KUKA KRL program: ps_r5_l_resp1_c1_mod.src, ps_r5_l_resp1_c1_mod.dat

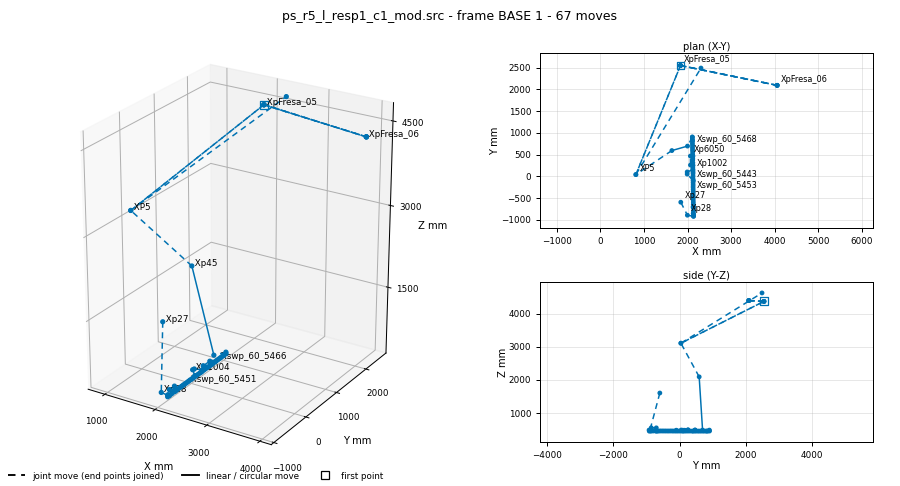
[picture p0: tool path of ps_r5_l_resp1_c1_mod.src in frame BASE 1, 67 of 69 moves have a stored position in this frame; points joined in program order, loops and branches not executed]
--- ps_r5_l_resp1_c1_mod.src ---
&ACCESS RVO1
&REL 40
&COMMENT C1 Respot LTA/LTB/MGS/MGSB
&PARAM DISKPATH = KRC:\R1\Program\SOLDA LTC
DEF ps_r5_l_resp1_c1_mod( )
;FOLD INI
  ;FOLD BASISTECH INI
    GLOBAL INTERRUPT DECL 3 WHEN $STOPMESS==TRUE DO IR_STOPM ( )
    INTERRUPT ON 3
    BAS (#INITMOV,0 )
  ;ENDFOLD (BASISTECH INI)
;FOLD SPOTTECH INI
USERSPOT(#INIT)
;ENDFOLD (SPOTTECH INI)
;FOLD GRIPPERTECH INI

;ENDFOLD (GRIPPERTECH INI)
  ;FOLD USER INI
    ;Make your modifications here

     ;FOLD COLLISION_V_3.01 INI ;%{E}
        IF (COLLISION_DATA[1].I_NR>0) THEN
          GLOBAL INTERRUPT DECL 21 WHEN $IN[COLLISION_DATA[1].I_NR]==FALSE DO COLLSTOP (1,0 )
        ENDIF
        IF (COLLISION_DATA[2].I_NR>0) THEN
          GLOBAL INTERRUPT DECL 22 WHEN $IN[COLLISION_DATA[2].I_NR]==FALSE DO COLLSTOP (2,0 )
        ENDIF
        IF (COLLISION_DATA[3].I_NR>0) THEN
          GLOBAL INTERRUPT DECL 23 WHEN $IN[COLLISION_DATA[3].I_NR]==FALSE DO COLLSTOP (3,0 )
        ENDIF
        IF (COLLISION_DATA[4].I_NR>0) THEN
          GLOBAL INTERRUPT DECL 24 WHEN $IN[COLLISION_DATA[4].I_NR]==FALSE DO COLLSTOP (4,0 )
        ENDIF
     ;ENDFOLD (Collision)

  ;ENDFOLD (USER INI)
;ENDFOLD (INI)

; Caracterização dos meios de produção: P13.060-R5
; Versão atual: 17/07/2013 Nome: Solda Respot C1
; Change: LTA/LTB/MGS/MGSB

chk_w2_wechs_ok ( )           ; VERIFICAÇÃO DE FERRAMENA: C1

;FOLD PTP HOME2 Vel=100 % DEFAULT;%{PE}%R 8.2.20,%MKUKATPBASIS,%CMOVE,%VPTP,%P 1:PTP, 2:HOME2, 3:, 5:100, 7:DEFAULT
$BWDSTART=FALSE
PDAT_ACT=PDEFAULT
FDAT_ACT=FHOME2
BAS(#PTP_PARAMS,100)
PTP XHOME2
;ENDFOLD

IF(NOT(GHOST())) THEN
IF MaxStandMenge (1) THEN
 MaxStandmengeErreicht (1)
ENDIF

IF Elektrodenwechsel (1) THEN
;FOLD PTP pFresa_05 CONT Vel=100 % PDAT40 Tool[2]:Gun C1 Base[1]:Actros;%{PE}%R 8.2.20,%MKUKATPBASIS,%CMOVE,%VPTP,%P 1:PTP, 2:pFresa_05, 3:C_DIS, 5:100, 7:PDAT40
$BWDSTART=FALSE
PDAT_ACT=PPDAT40
FDAT_ACT=FpFresa_05
BAS(#PTP_PARAMS,100)
PTP XpFresa_05 C_DIS
;ENDFOLD
;FOLD PULSE 168 'DOCK 1 Fechar Proteção' State=TRUE Time=1 sec;%{PE}%R 8.2.20,%MKUKATPBASIS,%COUT,%VPULSE,%P 2:168, 3:DOCK 1 Fechar Proteção, 5:TRUE, 6:, 8:1
PULSE($OUT[168], TRUE,1)
;ENDFOLD
;FOLD WAIT FOR ( IN 166 'DOCK 1 Proteção Fechada' );%{PE}%R 8.2.20,%MKUKATPBASIS,%CEXT_WAIT_FOR,%VEXT_WAIT_FOR,%P 2:, 4:, 5:$IN, 6:166, 7:DOCK 1 Proteção Fechada, 9:
WAIT FOR  ( $IN[166] )
;ENDFOLD
;FOLD PTP pFresa_06 CONT Vel=100 % PDAT41 Tool[2]:Gun C1 Base[1]:Actros;%{PE}%R 8.2.20,%MKUKATPBASIS,%CMOVE,%VPTP,%P 1:PTP, 2:pFresa_06, 3:C_DIS, 5:100, 7:PDAT41
$BWDSTART=FALSE
PDAT_ACT=PPDAT41
FDAT_ACT=FpFresa_06
BAS(#PTP_PARAMS,100)
PTP XpFresa_06 C_DIS
;ENDFOLD
 e_Fraes_2 ()
;FOLD PTP pFresa_07 CONT Vel=100 % PDAT42 Tool[2]:Gun C1 Base[1]:Actros;%{PE}%R 8.2.20,%MKUKATPBASIS,%CMOVE,%VPTP,%P 1:PTP, 2:pFresa_07, 3:C_DIS, 5:100, 7:PDAT42
$BWDSTART=FALSE
PDAT_ACT=PPDAT42
FDAT_ACT=FpFresa_07
BAS(#PTP_PARAMS,100)
PTP XpFresa_07 C_DIS
;ENDFOLD
;FOLD PTP pFresa_08 CONT Vel=100 % PDAT43 Tool[2]:Gun C1 Base[1]:Actros;%{PE}%R 8.2.20,%MKUKATPBASIS,%CMOVE,%VPTP,%P 1:PTP, 2:pFresa_08, 3:C_DIS, 5:100, 7:PDAT43
$BWDSTART=FALSE
PDAT_ACT=PPDAT43
FDAT_ACT=FpFresa_08
BAS(#PTP_PARAMS,100)
PTP XpFresa_08 C_DIS
;ENDFOLD
ENDIF
ENDIF
;FOLD PTP HOME2 Vel=100 % DEFAULT;%{PE}%R 8.2.20,%MKUKATPBASIS,%CMOVE,%VPTP,%P 1:PTP, 2:HOME2, 3:, 5:100, 7:DEFAULT
$BWDSTART=FALSE
PDAT_ACT=PDEFAULT
FDAT_ACT=FHOME2
BAS(#PTP_PARAMS,100)
PTP XHOME2
;ENDFOLD

;FOLD OUT 3339 'R5 SOLDANDO' State=TRUE ;%{PE}%R 8.2.20,%MKUKATPBASIS,%COUT,%VOUTX,%P 2:3339, 3:R5 SOLDANDO, 5:TRUE, 6:
$OUT[3339]=TRUE
;ENDFOLD
;FOLD OUT 3340 'locking-signal PLC' State=FALSE ;%{PE}%R 8.2.20,%MKUKATPBASIS,%COUT,%VOUTX,%P 2:3340, 3:locking-signal PLC, 5:FALSE, 6:
$OUT[3340]=FALSE
;ENDFOLD

;FOLD PTP p27 CONT Vel=100 % P_OLP2 Tool[2]:Gun C1 Base[1]:Actros;%{PE}%R 8.2.20,%MKUKATPBASIS,%CMOVE,%VPTP,%P 1:PTP, 2:p27, 3:C_DIS, 5:100, 7:P_OLP2
$BWDSTART=FALSE
PDAT_ACT=PP_OLP2
FDAT_ACT=Fp27
BAS(#PTP_PARAMS,100)
PTP Xp27 C_DIS
;ENDFOLD
;FOLD PTP p28 CONT Vel=100 % P_OLP3 Tool[2]:Gun C1 Base[1]:Actros;%{PE}%R 8.2.20,%MKUKATPBASIS,%CMOVE,%VPTP,%P 1:PTP, 2:p28, 3:C_DIS, 5:100, 7:P_OLP3
$BWDSTART=FALSE
PDAT_ACT=PP_OLP3
FDAT_ACT=Fp28
BAS(#PTP_PARAMS,100)
PTP Xp28 C_DIS
;ENDFOLD
;FOLD PTP p29 CONT Vel=100 % P_OLP4 Tool[2]:Gun C1 Base[1]:Actros;%{PE}%R8.2,%MKUKATPBASIS,%CMOVE,%VPTP,%P 1:PTP, 2:p29, 3:C_DIS, 5:100, 7:P_OLP4
$BWDSTART = FALSE
PDAT_ACT= PP_OLP4
FDAT_ACT= Fp29
BAS(#PTP_PARAMS,100)
PTP Xp29 C_DIS
;ENDFOLD

;FOLD ; SWP_60_5475;%{PE}%R 8.2.20,%MKUKATPBASIS,%CCOMMENT,%VNORMAL,%P 2:SWP_60_5475
;ENDFOLD
;FOLD PTP swp_60_5475 PDAT1 SPOT Gun=1 RETR OPN PgNo1=20 ACTIVE=1 Tool[2]:Gun C1 Base[1]:Actros;%{PE}%R 8.2.2,%MKUKATPSPOT,%CSPOT,%VPTP,%P 1:PTP, 2:swp_60_5475, 3:, 5:100, 7:PDAT1, 10:1, 12:#FIRST, 14:#OPN, 16:20, 18:1, 20:0, 22:0, 24:1, 25:NORMAL
$BWDSTART=FALSE
PDAT_ACT=PPDAT1
FDAT_ACT=Fswp_60_5475
BAS(#PTP_PARAMS,PPDAT1.VEL)
S_ACT.GUN=1
S_ACT.PAIR=SDEFAULT.PAIR
S_ACT.RETR=#OPN
S_ACT.CLO_TM=1
S_ACT.PGNO1=20
S_ACT.PGNO2=SDEFAULT.PGNO2
S_ACT.PRESS1=SDEFAULT.PRESS1
S_ACT.PRESS2=SDEFAULT.PRESS2
S_READY=FALSE
PTP Xswp_60_5475
USERSPOT(#SPOT, S_ACT)
WAIT FOR S_READY
;ENDFOLD
;FOLD PTP p6045 Vel=100 % PDAT48 Tool[2]:Gun C1 Base[1]:Actros;%{PE}%R 8.2.20,%MKUKATPBASIS,%CMOVE,%VPTP,%P 1:PTP, 2:p6045, 3:, 5:100, 7:PDAT48
$BWDSTART=FALSE
PDAT_ACT=PPDAT48
FDAT_ACT=Fp6045
BAS(#PTP_PARAMS,100)
PTP Xp6045
;ENDFOLD

;FOLD ; SWP_60_5473;%{PE}%R 8.2.20,%MKUKATPBASIS,%CCOMMENT,%VNORMAL,%P 2:SWP_60_5473
;ENDFOLD
;FOLD PTP swp_60_5473 PDAT2 SPOT Gun=1 RETR OPN PgNo1=21 ACTIVE=1 Tool[2]:Gun C1 Base[1]:Actros;%{PE}%R 8.2.2,%MKUKATPSPOT,%CSPOT,%VPTP,%P 1:PTP, 2:swp_60_5473, 3:, 5:100, 7:PDAT2, 10:1, 12:#FIRST, 14:#OPN, 16:21, 18:1, 20:0, 22:0, 24:1, 25:NORMAL
$BWDSTART=FALSE
PDAT_ACT=PPDAT2
FDAT_ACT=Fswp_60_5473
BAS(#PTP_PARAMS,PPDAT2.VEL)
S_ACT.GUN=1
S_ACT.PAIR=SDEFAULT.PAIR
S_ACT.RETR=#OPN
S_ACT.CLO_TM=1
S_ACT.PGNO1=21
S_ACT.PGNO2=SDEFAULT.PGNO2
S_ACT.PRESS1=SDEFAULT.PRESS1
S_ACT.PRESS2=SDEFAULT.PRESS2
S_READY=FALSE
PTP Xswp_60_5473
USERSPOT(#SPOT, S_ACT)
WAIT FOR S_READY
;ENDFOLD

; INSERCAO DO PONTO 60_5471 (ACTROS RETO_SEM BOLHA)
IF ($IN[3341]==TRUE) THEN

Wait for false
;FOLD ; Favor chamar a manutencao;%{PE}%R 8.2.20,%MKUKATPBASIS,%CCOMMENT,%VNORMAL,%P 2:Favor  chamar  a  manutencao
;ENDFOLD

;FOLD ; SWP_60_5471;%{PE}%R 8.2.20,%MKUKATPBASIS,%CCOMMENT,%VNORMAL,%P 2: SWP_60_5471
;ENDFOLD
;FOLD PTP swp_60_5477 P_OLP55 SPOT Gun=1 RETR OPN PgNo1=55 ACTIVE=1 Tool[2]:Gun C1 Base[1]:Actros;%{PE}%R 8.2.2,%MKUKATPSPOT,%CSPOT,%VPTP,%P 1:PTP, 2:swp_60_5477, 3:, 5:100, 7:P_OLP55, 10:1, 12:#FIRST, 14:#OPN, 16:55, 18:1, 20:1, 22:0, 24:1, 25:S_OLP1
$BWDSTART=FALSE
PDAT_ACT=PP_OLP55
FDAT_ACT=Fswp_60_5477
BAS(#PTP_PARAMS,PP_OLP55.VEL)
S_ACT.GUN=1
S_ACT.PAIR=SDEFAULT.PAIR
S_ACT.RETR=#OPN
S_ACT.CLO_TM=1
S_ACT.PGNO1=55
S_ACT.PGNO2=SDEFAULT.PGNO2
S_ACT.PRESS1=SDEFAULT.PRESS1
S_ACT.PRESS2=SDEFAULT.PRESS2
S_READY=FALSE
PTP Xswp_60_5477
USERSPOT(#SPOT, S_ACT)
WAIT FOR S_READY

;ENDFOLD
ENDIF

IF ($IN[3341]==FALSE) THEN
;FOLD PTP p30 CONT Vel=100 % P_OLP6 Tool[2]:Gun C1 Base[1]:Actros;%{PE}%R8.2,%MKUKATPBASIS,%CMOVE,%VPTP,%P 1:PTP, 2:p30, 3:C_DIS, 5:100, 7:P_OLP6
$BWDSTART = FALSE
PDAT_ACT= PP_OLP6
FDAT_ACT= Fp30
BAS(#PTP_PARAMS,100)
PTP Xp30 C_DIS
;ENDFOLD
;FOLD PTP p1005 CONT Vel=100 % DEFAULT Tool[2]:Gun C1 Base[1]:Actros;%{PE}%R 8.2.20,%MKUKATPBASIS,%CMOVE,%VPTP,%P 1:PTP, 2:p1005, 3:C_DIS, 5:100, 7:DEFAULT
$BWDSTART=FALSE
PDAT_ACT=PDEFAULT
FDAT_ACT=Fp1005
BAS(#PTP_PARAMS,100)
PTP Xp1005 C_DIS
;ENDFOLD
;FOLD PTP p31 CONT Vel=100 % P_OLP7 Tool[2]:Gun C1 Base[1]:Actros;%{PE}%R8.2,%MKUKATPBASIS,%CMOVE,%VPTP,%P 1:PTP, 2:p31, 3:C_DIS, 5:100, 7:P_OLP7
$BWDSTART = FALSE
PDAT_ACT= PP_OLP7
FDAT_ACT= Fp31
BAS(#PTP_PARAMS,100)
PTP Xp31 C_DIS
;ENDFOLD
ENDIF

;FOLD ; SWP_60_5469;%{PE}%R 8.2.20,%MKUKATPBASIS,%CCOMMENT,%VNORMAL,%P 2:SWP_60_5469
;ENDFOLD
;FOLD PTP swp_60_5469 PDAT3 SPOT Gun=1 RETR OPN PgNo1=22 ACTIVE=1 Tool[2]:Gun C1 Base[1]:Actros;%{PE}%R 8.2.2,%MKUKATPSPOT,%CSPOT,%VPTP,%P 1:PTP, 2:swp_60_5469, 3:, 5:100, 7:PDAT3, 10:1, 12:#FIRST, 14:#OPN, 16:22, 18:1, 20:0, 22:0, 24:1, 25:NORMAL
$BWDSTART=FALSE
PDAT_ACT=PPDAT3
FDAT_ACT=Fswp_60_5469
BAS(#PTP_PARAMS,PPDAT3.VEL)
S_ACT.GUN=1
S_ACT.PAIR=SDEFAULT.PAIR
S_ACT.RETR=#OPN
S_ACT.CLO_TM=1
S_ACT.PGNO1=22
S_ACT.PGNO2=SDEFAULT.PGNO2
S_ACT.PRESS1=SDEFAULT.PRESS1
S_ACT.PRESS2=SDEFAULT.PRESS2
S_READY=FALSE
PTP Xswp_60_5469
USERSPOT(#SPOT, S_ACT)
WAIT FOR S_READY
;ENDFOLD

;FOLD ; SWP_60_5467;%{PE}%R 8.2.20,%MKUKATPBASIS,%CCOMMENT,%VNORMAL,%P 2:SWP_60_5467
;ENDFOLD
;FOLD PTP swp_60_5467 PDAT4 SPOT Gun=1 RETR OPN PgNo1=23 ACTIVE=1 Tool[2]:Gun C1 Base[1]:Actros;%{PE}%R 8.2.2,%MKUKATPSPOT,%CSPOT,%VPTP,%P 1:PTP, 2:swp_60_5467, 3:, 5:100, 7:PDAT4, 10:1, 12:#FIRST, 14:#OPN, 16:23, 18:1, 20:0, 22:0, 24:1, 25:NORMAL
$BWDSTART=FALSE
PDAT_ACT=PPDAT4
FDAT_ACT=Fswp_60_5467
BAS(#PTP_PARAMS,PPDAT4.VEL)
S_ACT.GUN=1
S_ACT.PAIR=SDEFAULT.PAIR
S_ACT.RETR=#OPN
S_ACT.CLO_TM=1
S_ACT.PGNO1=23
S_ACT.PGNO2=SDEFAULT.PGNO2
S_ACT.PRESS1=SDEFAULT.PRESS1
S_ACT.PRESS2=SDEFAULT.PRESS2
S_READY=FALSE
PTP Xswp_60_5467
USERSPOT(#SPOT, S_ACT)
WAIT FOR S_READY
;ENDFOLD

;FOLD ; SWP_60_5465;%{PE}%R 8.2.20,%MKUKATPBASIS,%CCOMMENT,%VNORMAL,%P 2:SWP_60_5465
;ENDFOLD
;FOLD PTP swp_60_5465 PDAT5 SPOT Gun=1 RETR OPN PgNo1=24 ACTIVE=1 Tool[2]:Gun C1 Base[1]:Actros;%{PE}%R 8.2.2,%MKUKATPSPOT,%CSPOT,%VPTP,%P 1:PTP, 2:swp_60_5465, 3:, 5:100, 7:PDAT5, 10:1, 12:#FIRST, 14:#OPN, 16:24, 18:1, 20:0, 22:0, 24:1, 25:NORMAL
$BWDSTART=FALSE
PDAT_ACT=PPDAT5
FDAT_ACT=Fswp_60_5465
BAS(#PTP_PARAMS,PPDAT5.VEL)
S_ACT.GUN=1
S_ACT.PAIR=SDEFAULT.PAIR
S_ACT.RETR=#OPN
S_ACT.CLO_TM=1
S_ACT.PGNO1=24
S_ACT.PGNO2=SDEFAULT.PGNO2
S_ACT.PRESS1=SDEFAULT.PRESS1
S_ACT.PRESS2=SDEFAULT.PRESS2
S_READY=FALSE
PTP Xswp_60_5465
USERSPOT(#SPOT, S_ACT)
WAIT FOR S_READY
;ENDFOLD

;FOLD ; SWP_60_5463;%{PE}%R 8.2.20,%MKUKATPBASIS,%CCOMMENT,%VNORMAL,%P 2:SWP_60_5463
;ENDFOLD
;FOLD PTP swp_60_5463 PDAT6 SPOT Gun=1 RETR OPN PgNo1=25 ACTIVE=1 Tool[2]:Gun C1 Base[1]:Actros;%{PE}%R 8.2.2,%MKUKATPSPOT,%CSPOT,%VPTP,%P 1:PTP, 2:swp_60_5463, 3:, 5:100, 7:PDAT6, 10:1, 12:#FIRST, 14:#OPN, 16:25, 18:1, 20:0, 22:0, 24:1, 25:NORMAL
$BWDSTART=FALSE
PDAT_ACT=PPDAT6
FDAT_ACT=Fswp_60_5463
BAS(#PTP_PARAMS,PPDAT6.VEL)
S_ACT.GUN=1
S_ACT.PAIR=SDEFAULT.PAIR
S_ACT.RETR=#OPN
S_ACT.CLO_TM=1
S_ACT.PGNO1=25
S_ACT.PGNO2=SDEFAULT.PGNO2
S_ACT.PRESS1=SDEFAULT.PRESS1
S_ACT.PRESS2=SDEFAULT.PRESS2
S_READY=FALSE
PTP Xswp_60_5463
USERSPOT(#SPOT, S_ACT)
WAIT FOR S_READY
;ENDFOLD

;FOLD ; SWP_60_5461;%{PE}%R 8.2.20,%MKUKATPBASIS,%CCOMMENT,%VNORMAL,%P 2:SWP_60_5461
;ENDFOLD
;FOLD PTP swp_60_5461 PDAT7 SPOT Gun=1 RETR OPN PgNo1=26 ACTIVE=1 Tool[2]:Gun C1 Base[1]:Actros;%{PE}%R 8.2.2,%MKUKATPSPOT,%CSPOT,%VPTP,%P 1:PTP, 2:swp_60_5461, 3:, 5:100, 7:PDAT7, 10:1, 12:#FIRST, 14:#OPN, 16:26, 18:1, 20:0, 22:0, 24:1, 25:NORMAL
$BWDSTART=FALSE
PDAT_ACT=PPDAT7
FDAT_ACT=Fswp_60_5461
BAS(#PTP_PARAMS,PPDAT7.VEL)
S_ACT.GUN=1
S_ACT.PAIR=SDEFAULT.PAIR
S_ACT.RETR=#OPN
S_ACT.CLO_TM=1
S_ACT.PGNO1=26
S_ACT.PGNO2=SDEFAULT.PGNO2
S_ACT.PRESS1=SDEFAULT.PRESS1
S_ACT.PRESS2=SDEFAULT.PRESS2
S_READY=FALSE
PTP Xswp_60_5461
USERSPOT(#SPOT, S_ACT)
WAIT FOR S_READY
;ENDFOLD

;FOLD ; SWP_60_5459;%{PE}%R 8.2.20,%MKUKATPBASIS,%CCOMMENT,%VNORMAL,%P 2:SWP_60_5459
;ENDFOLD
;FOLD PTP swp_60_5459 PDAT8 SPOT Gun=1 RETR OPN PgNo1=27 ACTIVE=1 Tool[2]:Gun C1 Base[1]:Actros;%{PE}%R 8.2.2,%MKUKATPSPOT,%CSPOT,%VPTP,%P 1:PTP, 2:swp_60_5459, 3:, 5:100, 7:PDAT8, 10:1, 12:#FIRST, 14:#OPN, 16:27, 18:1, 20:0, 22:0, 24:1, 25:NORMAL
$BWDSTART=FALSE
PDAT_ACT=PPDAT8
FDAT_ACT=Fswp_60_5459
BAS(#PTP_PARAMS,PPDAT8.VEL)
S_ACT.GUN=1
S_ACT.PAIR=SDEFAULT.PAIR
S_ACT.RETR=#OPN
S_ACT.CLO_TM=1
S_ACT.PGNO1=27
S_ACT.PGNO2=SDEFAULT.PGNO2
S_ACT.PRESS1=SDEFAULT.PRESS1
S_ACT.PRESS2=SDEFAULT.PRESS2
S_READY=FALSE
PTP Xswp_60_5459
USERSPOT(#SPOT, S_ACT)
WAIT FOR S_READY
;ENDFOLD

;FOLD ; SWP_60_5457;%{PE}%R 8.2.20,%MKUKATPBASIS,%CCOMMENT,%VNORMAL,%P 2:SWP_60_5457
;ENDFOLD
;FOLD PTP swp_60_5457 PDAT9 SPOT Gun=1 RETR OPN PgNo1=28 ACTIVE=1 Tool[2]:Gun C1 Base[1]:Actros;%{PE}%R 8.2.2,%MKUKATPSPOT,%CSPOT,%VPTP,%P 1:PTP, 2:swp_60_5457, 3:, 5:100, 7:PDAT9, 10:1, 12:#FIRST, 14:#OPN, 16:28, 18:1, 20:0, 22:0, 24:1, 25:NORMAL
$BWDSTART=FALSE
PDAT_ACT=PPDAT9
FDAT_ACT=Fswp_60_5457
BAS(#PTP_PARAMS,PPDAT9.VEL)
S_ACT.GUN=1
S_ACT.PAIR=SDEFAULT.PAIR
S_ACT.RETR=#OPN
S_ACT.CLO_TM=1
S_ACT.PGNO1=28
S_ACT.PGNO2=SDEFAULT.PGNO2
S_ACT.PRESS1=SDEFAULT.PRESS1
S_ACT.PRESS2=SDEFAULT.PRESS2
S_READY=FALSE
PTP Xswp_60_5457
USERSPOT(#SPOT, S_ACT)
WAIT FOR S_READY
;ENDFOLD

;FOLD ; SWP_60_5455;%{PE}%R 8.2.20,%MKUKATPBASIS,%CCOMMENT,%VNORMAL,%P 2:SWP_60_5455
;ENDFOLD
;FOLD PTP swp_60_5455 PDAT10 SPOT Gun=1 RETR OPN PgNo1=29 ACTIVE=1 Tool[2]:Gun C1 Base[1]:Actros;%{PE}%R 8.2.2,%MKUKATPSPOT,%CSPOT,%VPTP,%P 1:PTP, 2:swp_60_5455, 3:, 5:100, 7:PDAT10, 10:1, 12:#FIRST, 14:#OPN, 16:29, 18:1, 20:0, 22:0, 24:1, 25:NORMAL
$BWDSTART=FALSE
PDAT_ACT=PPDAT10
FDAT_ACT=Fswp_60_5455
BAS(#PTP_PARAMS,PPDAT10.VEL)
S_ACT.GUN=1
S_ACT.PAIR=SDEFAULT.PAIR
S_ACT.RETR=#OPN
S_ACT.CLO_TM=1
S_ACT.PGNO1=29
S_ACT.PGNO2=SDEFAULT.PGNO2
S_ACT.PRESS1=SDEFAULT.PRESS1
S_ACT.PRESS2=SDEFAULT.PRESS2
S_READY=FALSE
PTP Xswp_60_5455
USERSPOT(#SPOT, S_ACT)
WAIT FOR S_READY
;ENDFOLD

;FOLD ; SWP_60_5453;%{PE}%R 8.2.20,%MKUKATPBASIS,%CCOMMENT,%VNORMAL,%P 2:SWP_60_5453
;ENDFOLD
;FOLD PTP swp_60_5453 PDAT11 SPOT Gun=1 RETR OPN PgNo1=30 ACTIVE=1 Tool[2]:Gun C1 Base[1]:Actros;%{PE}%R 8.2.2,%MKUKATPSPOT,%CSPOT,%VPTP,%P 1:PTP, 2:swp_60_5453, 3:, 5:100, 7:PDAT11, 10:1, 12:#FIRST, 14:#OPN, 16:30, 18:1, 20:0, 22:0, 24:1, 25:NORMAL
$BWDSTART=FALSE
PDAT_ACT=PPDAT11
FDAT_ACT=Fswp_60_5453
BAS(#PTP_PARAMS,PPDAT11.VEL)
S_ACT.GUN=1
S_ACT.PAIR=SDEFAULT.PAIR
S_ACT.RETR=#OPN
S_ACT.CLO_TM=1
S_ACT.PGNO1=30
S_ACT.PGNO2=SDEFAULT.PGNO2
S_ACT.PRESS1=SDEFAULT.PRESS1
S_ACT.PRESS2=SDEFAULT.PRESS2
S_READY=FALSE
PTP Xswp_60_5453
USERSPOT(#SPOT, S_ACT)
WAIT FOR S_READY
;ENDFOLD

;FOLD ; SWP_60_5451;%{PE}%R 8.2.20,%MKUKATPBASIS,%CCOMMENT,%VNORMAL,%P 2:SWP_60_5451
;ENDFOLD
;FOLD PTP swp_60_5451 PDAT12 SPOT Gun=1 RETR OPN PgNo1=31 ACTIVE=1 Tool[2]:Gun C1 Base[1]:Actros;%{PE}%R 8.2.2,%MKUKATPSPOT,%CSPOT,%VPTP,%P 1:PTP, 2:swp_60_5451, 3:, 5:100, 7:PDAT12, 10:1, 12:#FIRST, 14:#OPN, 16:31, 18:1, 20:0, 22:0, 24:1, 25:NORMAL
$BWDSTART=FALSE
PDAT_ACT=PPDAT12
FDAT_ACT=Fswp_60_5451
BAS(#PTP_PARAMS,PPDAT12.VEL)
S_ACT.GUN=1
S_ACT.PAIR=SDEFAULT.PAIR
S_ACT.RETR=#OPN
S_ACT.CLO_TM=1
S_ACT.PGNO1=31
S_ACT.PGNO2=SDEFAULT.PGNO2
S_ACT.PRESS1=SDEFAULT.PRESS1
S_ACT.PRESS2=SDEFAULT.PRESS2
S_READY=FALSE
PTP Xswp_60_5451
USERSPOT(#SPOT, S_ACT)
WAIT FOR S_READY
;ENDFOLD

;FOLD ; SWP_60_5449;%{PE}%R 8.2.20,%MKUKATPBASIS,%CCOMMENT,%VNORMAL,%P 2:SWP_60_5449
;ENDFOLD
;FOLD PTP swp_60_5449 PDAT13 SPOT Gun=1 RETR OPN PgNo1=32 ACTIVE=1 Tool[2]:Gun C1 Base[1]:Actros;%{PE}%R 8.2.2,%MKUKATPSPOT,%CSPOT,%VPTP,%P 1:PTP, 2:swp_60_5449, 3:, 5:100, 7:PDAT13, 10:1, 12:#FIRST, 14:#OPN, 16:32, 18:1, 20:0, 22:0, 24:1, 25:NORMAL
$BWDSTART=FALSE
PDAT_ACT=PPDAT13
FDAT_ACT=Fswp_60_5449
BAS(#PTP_PARAMS,PPDAT13.VEL)
S_ACT.GUN=1
S_ACT.PAIR=SDEFAULT.PAIR
S_ACT.RETR=#OPN
S_ACT.CLO_TM=1
S_ACT.PGNO1=32
S_ACT.PGNO2=SDEFAULT.PGNO2
S_ACT.PRESS1=SDEFAULT.PRESS1
S_ACT.PRESS2=SDEFAULT.PRESS2
S_READY=FALSE
PTP Xswp_60_5449
USERSPOT(#SPOT, S_ACT)
WAIT FOR S_READY
;ENDFOLD

;FOLD ; SWP_60_5447;%{PE}%R 8.2.20,%MKUKATPBASIS,%CCOMMENT,%VNORMAL,%P 2:SWP_60_5447
;ENDFOLD
;FOLD PTP swp_60_5447 PDAT14 SPOT Gun=1 RETR OPN PgNo1=33 ACTIVE=1 Tool[2]:Gun C1 Base[1]:Actros;%{PE}%R 8.2.2,%MKUKATPSPOT,%CSPOT,%VPTP,%P 1:PTP, 2:swp_60_5447, 3:, 5:100, 7:PDAT14, 10:1, 12:#FIRST, 14:#OPN, 16:33, 18:1, 20:0, 22:0, 24:1, 25:NORMAL
$BWDSTART=FALSE
PDAT_ACT=PPDAT14
FDAT_ACT=Fswp_60_5447
BAS(#PTP_PARAMS,PPDAT14.VEL)
S_ACT.GUN=1
S_ACT.PAIR=SDEFAULT.PAIR
S_ACT.RETR=#OPN
S_ACT.CLO_TM=1
S_ACT.PGNO1=33
S_ACT.PGNO2=SDEFAULT.PGNO2
S_ACT.PRESS1=SDEFAULT.PRESS1
S_ACT.PRESS2=SDEFAULT.PRESS2
S_READY=FALSE
PTP Xswp_60_5447
USERSPOT(#SPOT, S_ACT)
WAIT FOR S_READY
;ENDFOLD

;FOLD ; SWP_60_5445;%{PE}%R 8.2.20,%MKUKATPBASIS,%CCOMMENT,%VNORMAL,%P 2:SWP_60_5445
;ENDFOLD
;FOLD PTP swp_60_5445 PDAT15 SPOT Gun=1 RETR OPN PgNo1=34 ACTIVE=1 Tool[2]:Gun C1 Base[1]:Actros;%{PE}%R 8.2.2,%MKUKATPSPOT,%CSPOT,%VPTP,%P 1:PTP, 2:swp_60_5445, 3:, 5:100, 7:PDAT15, 10:1, 12:#FIRST, 14:#OPN, 16:34, 18:1, 20:0, 22:0, 24:1, 25:NORMAL
$BWDSTART=FALSE
PDAT_ACT=PPDAT15
FDAT_ACT=Fswp_60_5445
BAS(#PTP_PARAMS,PPDAT15.VEL)
S_ACT.GUN=1
S_ACT.PAIR=SDEFAULT.PAIR
S_ACT.RETR=#OPN
S_ACT.CLO_TM=1
S_ACT.PGNO1=34
S_ACT.PGNO2=SDEFAULT.PGNO2
S_ACT.PRESS1=SDEFAULT.PRESS1
S_ACT.PRESS2=SDEFAULT.PRESS2
S_READY=FALSE
PTP Xswp_60_5445
USERSPOT(#SPOT, S_ACT)
WAIT FOR S_READY
;ENDFOLD

;FOLD ; SWP_60_5443;%{PE}%R 8.2.20,%MKUKATPBASIS,%CCOMMENT,%VNORMAL,%P 2:SWP_60_5443
;ENDFOLD
;FOLD PTP swp_60_5443 PDAT16 SPOT Gun=1 RETR OPN PgNo1=35 ACTIVE=1 Tool[2]:Gun C1 Base[1]:Actros;%{PE}%R 8.2.2,%MKUKATPSPOT,%CSPOT,%VPTP,%P 1:PTP, 2:swp_60_5443, 3:, 5:100, 7:PDAT16, 10:1, 12:#FIRST, 14:#OPN, 16:35, 18:1, 20:0, 22:0, 24:1, 25:NORMAL
$BWDSTART=FALSE
PDAT_ACT=PPDAT16
FDAT_ACT=Fswp_60_5443
BAS(#PTP_PARAMS,PPDAT16.VEL)
S_ACT.GUN=1
S_ACT.PAIR=SDEFAULT.PAIR
S_ACT.RETR=#OPN
S_ACT.CLO_TM=1
S_ACT.PGNO1=35
S_ACT.PGNO2=SDEFAULT.PGNO2
S_ACT.PRESS1=SDEFAULT.PRESS1
S_ACT.PRESS2=SDEFAULT.PRESS2
S_READY=FALSE
PTP Xswp_60_5443
USERSPOT(#SPOT, S_ACT)
WAIT FOR S_READY
;ENDFOLD

;FOLD ; SWP_60_5441;%{PE}%R 8.2.20,%MKUKATPBASIS,%CCOMMENT,%VNORMAL,%P 2:SWP_60_5441
;ENDFOLD
;FOLD PTP p60_5441 DEFAULT SPOT Gun=1 RETR OPN PgNo1=36 ACTIVE=1 Tool[2]:Gun C1 Base[1]:Actros;%{PE}%R 8.2.2,%MKUKATPSPOT,%CSPOT,%VPTP,%P 1:PTP, 2:p60_5441, 3:, 5:100, 7:DEFAULT, 10:1, 12:#FIRST, 14:#OPN, 16:36, 18:1, 20:0, 22:0, 24:1, 25:NORMAL
$BWDSTART=FALSE
PDAT_ACT=PDEFAULT
FDAT_ACT=Fp60_5441
BAS(#PTP_PARAMS,PDEFAULT.VEL)
S_ACT.GUN=1
S_ACT.PAIR=SDEFAULT.PAIR
S_ACT.RETR=#OPN
S_ACT.CLO_TM=1
S_ACT.PGNO1=36
S_ACT.PGNO2=SDEFAULT.PGNO2
S_ACT.PRESS1=SDEFAULT.PRESS1
S_ACT.PRESS2=SDEFAULT.PRESS2
S_READY=FALSE
PTP Xp60_5441
USERSPOT(#SPOT, S_ACT)
WAIT FOR S_READY
;ENDFOLD

; INSECAO DO PONTO 60_5497
IF ($IN[3342]==TRUE) THEN
;FOLD ; SWP 60_5497;%{PE}%R 8.2.20,%MKUKATPBASIS,%CCOMMENT,%VNORMAL,%P 2:SWP  60_5497
;ENDFOLD
;FOLD PTP swp_60_5497 PDAT55 SPOT Gun=1 RETR OPN PgNo1=37 ACTIVE=1 Tool[2]:Gun C1 Base[1]:Actros;%{PE}%R 8.2.2,%MKUKATPSPOT,%CSPOT,%VPTP,%P 1:PTP, 2:swp_60_5497, 3:, 5:100, 7:PDAT55, 10:1, 12:#FIRST, 14:#OPN, 16:37, 18:1, 20:0, 22:0, 24:1, 25:NORMAL
$BWDSTART=FALSE
PDAT_ACT=PPDAT55
FDAT_ACT=Fswp_60_5497
BAS(#PTP_PARAMS,PPDAT55.VEL)
S_ACT.GUN=1
S_ACT.PAIR=SDEFAULT.PAIR
S_ACT.RETR=#OPN
S_ACT.CLO_TM=1
S_ACT.PGNO1=37
S_ACT.PGNO2=SDEFAULT.PGNO2
S_ACT.PRESS1=SDEFAULT.PRESS1
S_ACT.PRESS2=SDEFAULT.PRESS2
S_READY=FALSE
PTP Xswp_60_5497
USERSPOT(#SPOT, S_ACT)
WAIT FOR S_READY
;ENDFOLD
ENDIF

IF ($IN[3342]==FALSE) THEN
;FOLD PTP p1003 CONT Vel=100 % DEFAULT Tool[2]:Gun C1 Base[1]:Actros;%{PE}%R 8.2.20,%MKUKATPBASIS,%CMOVE,%VPTP,%P 1:PTP, 2:p1003, 3:C_DIS, 5:100, 7:DEFAULT
$BWDSTART=FALSE
PDAT_ACT=PDEFAULT
FDAT_ACT=Fp1003
BAS(#PTP_PARAMS,100)
PTP Xp1003 C_DIS
;ENDFOLD
;FOLD PTP p1004 CONT Vel=100 % DEFAULT Tool[2]:Gun C1 Base[1]:Actros;%{PE}%R 8.2.20,%MKUKATPBASIS,%CMOVE,%VPTP,%P 1:PTP, 2:p1004, 3:C_DIS, 5:100, 7:DEFAULT
$BWDSTART=FALSE
PDAT_ACT=PDEFAULT
FDAT_ACT=Fp1004
BAS(#PTP_PARAMS,100)
PTP Xp1004 C_DIS
;ENDFOLD
;FOLD PTP p6044 CONT Vel=100 % DEFAULT Tool[2]:Gun C1 Base[1]:Actros;%{PE}%R 8.2.20,%MKUKATPBASIS,%CMOVE,%VPTP,%P 1:PTP, 2:p6044, 3:C_DIS, 5:100, 7:DEFAULT
$BWDSTART=FALSE
PDAT_ACT=PDEFAULT
FDAT_ACT=Fp6044
BAS(#PTP_PARAMS,100)
PTP Xp6044 C_DIS
;ENDFOLD
;FOLD PTP p1002 CONT Vel=100 % DEFAULT Tool[2]:Gun C1 Base[1]:Actros;%{PE}%R 8.2.20,%MKUKATPBASIS,%CMOVE,%VPTP,%P 1:PTP, 2:p1002, 3:C_DIS, 5:100, 7:DEFAULT
$BWDSTART=FALSE
PDAT_ACT=PDEFAULT
FDAT_ACT=Fp1002
BAS(#PTP_PARAMS,100)
PTP Xp1002 C_DIS
;ENDFOLD
ENDIF

;FOLD ; SWP_60_5442;%{PE}%R 8.2.20,%MKUKATPBASIS,%CCOMMENT,%VNORMAL,%P 2:SWP_60_5442
;ENDFOLD
;FOLD PTP swp_60_5442 PDAT51 SPOT Gun=1 RETR OPN PgNo1=37 ACTIVE=1 Tool[2]:Gun C1 Base[1]:Actros;%{PE}%R 8.2.2,%MKUKATPSPOT,%CSPOT,%VPTP,%P 1:PTP, 2:swp_60_5442, 3:, 5:100, 7:PDAT51, 10:1, 12:#FIRST, 14:#OPN, 16:37, 18:1, 20:0, 22:0, 24:1, 25:NORMAL
$BWDSTART=FALSE
PDAT_ACT=PPDAT51
FDAT_ACT=Fswp_60_5442
BAS(#PTP_PARAMS,PPDAT51.VEL)
S_ACT.GUN=1
S_ACT.PAIR=SDEFAULT.PAIR
S_ACT.RETR=#OPN
S_ACT.CLO_TM=1
S_ACT.PGNO1=37
S_ACT.PGNO2=SDEFAULT.PGNO2
S_ACT.PRESS1=SDEFAULT.PRESS1
S_ACT.PRESS2=SDEFAULT.PRESS2
S_READY=FALSE
PTP Xswp_60_5442
USERSPOT(#SPOT, S_ACT)
WAIT FOR S_READY
;ENDFOLD

;FOLD ; SWP_60_5444;%{PE}%R 8.2.20,%MKUKATPBASIS,%CCOMMENT,%VNORMAL,%P 2:SWP_60_5444
;ENDFOLD
;FOLD PTP swp_60_5444 PDAT19 SPOT Gun=1 RETR OPN PgNo1=38 ACTIVE=1 Tool[2]:Gun C1 Base[1]:Actros;%{PE}%R 8.2.2,%MKUKATPSPOT,%CSPOT,%VPTP,%P 1:PTP, 2:swp_60_5444, 3:, 5:100, 7:PDAT19, 10:1, 12:#FIRST, 14:#OPN, 16:38, 18:1, 20:0, 22:0, 24:1, 25:NORMAL
$BWDSTART=FALSE
PDAT_ACT=PPDAT19
FDAT_ACT=Fswp_60_5444
BAS(#PTP_PARAMS,PPDAT19.VEL)
S_ACT.GUN=1
S_ACT.PAIR=SDEFAULT.PAIR
S_ACT.RETR=#OPN
S_ACT.CLO_TM=1
S_ACT.PGNO1=38
S_ACT.PGNO2=SDEFAULT.PGNO2
S_ACT.PRESS1=SDEFAULT.PRESS1
S_ACT.PRESS2=SDEFAULT.PRESS2
S_READY=FALSE
PTP Xswp_60_5444
USERSPOT(#SPOT, S_ACT)
WAIT FOR S_READY
;ENDFOLD

;FOLD ; SWP_60_5446;%{PE}%R 8.2.20,%MKUKATPBASIS,%CCOMMENT,%VNORMAL,%P 2:SWP_60_5446
;ENDFOLD
;FOLD PTP swp_60_5446 PDAT20 SPOT Gun=1 RETR OPN PgNo1=39 ACTIVE=1 Tool[2]:Gun C1 Base[1]:Actros;%{PE}%R 8.2.2,%MKUKATPSPOT,%CSPOT,%VPTP,%P 1:PTP, 2:swp_60_5446, 3:, 5:100, 7:PDAT20, 10:1, 12:#FIRST, 14:#OPN, 16:39, 18:1, 20:0, 22:0, 24:1, 25:NORMAL
$BWDSTART=FALSE
PDAT_ACT=PPDAT20
FDAT_ACT=Fswp_60_5446
BAS(#PTP_PARAMS,PPDAT20.VEL)
S_ACT.GUN=1
S_ACT.PAIR=SDEFAULT.PAIR
S_ACT.RETR=#OPN
S_ACT.CLO_TM=1
S_ACT.PGNO1=39
S_ACT.PGNO2=SDEFAULT.PGNO2
S_ACT.PRESS1=SDEFAULT.PRESS1
S_ACT.PRESS2=SDEFAULT.PRESS2
S_READY=FALSE
PTP Xswp_60_5446
USERSPOT(#SPOT, S_ACT)
WAIT FOR S_READY
;ENDFOLD

;FOLD ; SWP_60_5448;%{PE}%R 8.2.20,%MKUKATPBASIS,%CCOMMENT,%VNORMAL,%P 2:SWP_60_5448
;ENDFOLD
;FOLD PTP swp_60_5448 PDAT21 SPOT Gun=1 RETR OPN PgNo1=40 ACTIVE=1 Tool[2]:Gun C1 Base[1]:Actros;%{PE}%R 8.2.2,%MKUKATPSPOT,%CSPOT,%VPTP,%P 1:PTP, 2:swp_60_5448, 3:, 5:100, 7:PDAT21, 10:1, 12:#FIRST, 14:#OPN, 16:40, 18:1, 20:0, 22:0, 24:1, 25:NORMAL
$BWDSTART=FALSE
PDAT_ACT=PPDAT21
FDAT_ACT=Fswp_60_5448
BAS(#PTP_PARAMS,PPDAT21.VEL)
S_ACT.GUN=1
S_ACT.PAIR=SDEFAULT.PAIR
S_ACT.RETR=#OPN
S_ACT.CLO_TM=1
S_ACT.PGNO1=40
S_ACT.PGNO2=SDEFAULT.PGNO2
S_ACT.PRESS1=SDEFAULT.PRESS1
S_ACT.PRESS2=SDEFAULT.PRESS2
S_READY=FALSE
PTP Xswp_60_5448
USERSPOT(#SPOT, S_ACT)
WAIT FOR S_READY
;ENDFOLD

;FOLD ; SWP_60_5450;%{PE}%R 8.2.20,%MKUKATPBASIS,%CCOMMENT,%VNORMAL,%P 2:SWP_60_5450
;ENDFOLD
;FOLD PTP swp_60_5450 PDAT22 SPOT Gun=1 RETR OPN PgNo1=41 ACTIVE=1 Tool[2]:Gun C1 Base[1]:Actros;%{PE}%R 8.2.2,%MKUKATPSPOT,%CSPOT,%VPTP,%P 1:PTP, 2:swp_60_5450, 3:, 5:100, 7:PDAT22, 10:1, 12:#FIRST, 14:#OPN, 16:41, 18:1, 20:0, 22:0, 24:1, 25:NORMAL
$BWDSTART=FALSE
PDAT_ACT=PPDAT22
FDAT_ACT=Fswp_60_5450
BAS(#PTP_PARAMS,PPDAT22.VEL)
S_ACT.GUN=1
S_ACT.PAIR=SDEFAULT.PAIR
S_ACT.RETR=#OPN
S_ACT.CLO_TM=1
S_ACT.PGNO1=41
S_ACT.PGNO2=SDEFAULT.PGNO2
S_ACT.PRESS1=SDEFAULT.PRESS1
S_ACT.PRESS2=SDEFAULT.PRESS2
S_READY=FALSE
PTP Xswp_60_5450
USERSPOT(#SPOT, S_ACT)
WAIT FOR S_READY
;ENDFOLD

; INSERCAO DO PONTO 60_5478 (ACTROS RETO_SEM BOLHA)
IF ($IN[3341]) THEN

Wait for false
;FOLD ; Favor chamar a manutencao;%{PE}%R 8.2.20,%MKUKATPBASIS,%CCOMMENT,%VNORMAL,%P 2:Favor  chamar  a  manutencao
;ENDFOLD

;FOLD ; SWP_60_5478;%{PE}%R 8.2.20,%MKUKATPBASIS,%CCOMMENT,%VNORMAL,%P 2:SWP_60_5478
;ENDFOLD
;FOLD PTP swp_60_5478 P_OLP56 SPOT Gun=1 RETR OPN PgNo1=56 ACTIVE=1 Tool[2]:Gun C1 Base[1]:Actros;%{PE}%R 8.2.2,%MKUKATPSPOT,%CSPOT,%VPTP,%P 1:PTP, 2:swp_60_5478, 3:, 5:100, 7:P_OLP56, 10:1, 12:#FIRST, 14:#OPN, 16:56, 18:1, 20:1, 22:0, 24:1, 25:S_OLP2
$BWDSTART=FALSE
PDAT_ACT=PP_OLP56
FDAT_ACT=Fswp_60_5478
BAS(#PTP_PARAMS,PP_OLP56.VEL)
S_ACT.GUN=1
S_ACT.PAIR=SDEFAULT.PAIR
S_ACT.RETR=#OPN
S_ACT.CLO_TM=1
S_ACT.PGNO1=56
S_ACT.PGNO2=SDEFAULT.PGNO2
S_ACT.PRESS1=SDEFAULT.PRESS1
S_ACT.PRESS2=SDEFAULT.PRESS2
S_READY=FALSE
PTP Xswp_60_5478
USERSPOT(#SPOT, S_ACT)
WAIT FOR S_READY

;ENDFOLD
ENDIF

IF (NOT $IN[3341]) THEN
;FOLD PTP p6046 CONT Vel=100 % PDAT49 Tool[2]:Gun C1 Base[1]:Actros;%{PE}%R 8.2.20,%MKUKATPBASIS,%CMOVE,%VPTP,%P 1:PTP, 2:p6046, 3:C_DIS, 5:100, 7:PDAT49
$BWDSTART=FALSE
PDAT_ACT=PPDAT49
FDAT_ACT=Fp6046
BAS(#PTP_PARAMS,100)
PTP Xp6046 C_DIS
;ENDFOLD
;FOLD PTP p6049 CONT Vel=100 % PDAT52 Tool[2]:Gun C1 Base[1]:Actros;%{PE}%R 8.2.20,%MKUKATPBASIS,%CMOVE,%VPTP,%P 1:PTP, 2:p6049, 3:C_DIS, 5:100, 7:PDAT52
$BWDSTART=FALSE
PDAT_ACT=PPDAT52
FDAT_ACT=Fp6049
BAS(#PTP_PARAMS,100)
PTP Xp6049 C_DIS
;ENDFOLD
;FOLD PTP p6050 CONT Vel=100 % PDAT53 Tool[2]:Gun C1 Base[1]:Actros;%{PE}%R 8.2.20,%MKUKATPBASIS,%CMOVE,%VPTP,%P 1:PTP, 2:p6050, 3:C_DIS, 5:100, 7:PDAT53
$BWDSTART=FALSE
PDAT_ACT=PPDAT53
FDAT_ACT=Fp6050
BAS(#PTP_PARAMS,100)
PTP Xp6050 C_DIS
;ENDFOLD
;FOLD PTP p6051 CONT Vel=100 % PDAT54 Tool[2]:Gun C1 Base[1]:Actros;%{PE}%R 8.2.20,%MKUKATPBASIS,%CMOVE,%VPTP,%P 1:PTP, 2:p6051, 3:C_DIS, 5:100, 7:PDAT54
$BWDSTART=FALSE
PDAT_ACT=PPDAT54
FDAT_ACT=Fp6051
BAS(#PTP_PARAMS,100)
PTP Xp6051 C_DIS
;ENDFOLD
ENDIF

;FOLD ; SWP_60_5454;%{PE}%R 8.2.20,%MKUKATPBASIS,%CCOMMENT,%VNORMAL,%P 2:SWP_60_5454
;ENDFOLD
;FOLD PTP swp_60_5454 PDAT24 SPOT Gun=1 RETR OPN PgNo1=42 ACTIVE=1 Tool[2]:Gun C1 Base[1]:Actros;%{PE}%R 8.2.2,%MKUKATPSPOT,%CSPOT,%VPTP,%P 1:PTP, 2:swp_60_5454, 3:, 5:100, 7:PDAT24, 10:1, 12:#FIRST, 14:#OPN, 16:42, 18:1, 20:0, 22:0, 24:1, 25:NORMAL
$BWDSTART=FALSE
PDAT_ACT=PPDAT24
FDAT_ACT=Fswp_60_5454
BAS(#PTP_PARAMS,PPDAT24.VEL)
S_ACT.GUN=1
S_ACT.PAIR=SDEFAULT.PAIR
S_ACT.RETR=#OPN
S_ACT.CLO_TM=1
S_ACT.PGNO1=42
S_ACT.PGNO2=SDEFAULT.PGNO2
S_ACT.PRESS1=SDEFAULT.PRESS1
S_ACT.PRESS2=SDEFAULT.PRESS2
S_READY=FALSE
PTP Xswp_60_5454
USERSPOT(#SPOT, S_ACT)
WAIT FOR S_READY
;ENDFOLD

;FOLD ; SWP_60_5456;%{PE}%R 8.2.20,%MKUKATPBASIS,%CCOMMENT,%VNORMAL,%P 2:SWP_60_5456
;ENDFOLD
;FOLD PTP swp_60_5456 PDAT25 SPOT Gun=1 RETR OPN PgNo1=43 ACTIVE=1 Tool[2]:Gun C1 Base[1]:Actros;%{PE}%R 8.2.2,%MKUKATPSPOT,%CSPOT,%VPTP,%P 1:PTP, 2:swp_60_5456, 3:, 5:100, 7:PDAT25, 10:1, 12:#FIRST, 14:#OPN, 16:43, 18:1, 20:0, 22:0, 24:1, 25:NORMAL
$BWDSTART=FALSE
PDAT_ACT=PPDAT25
FDAT_ACT=Fswp_60_5456
BAS(#PTP_PARAMS,PPDAT25.VEL)
S_ACT.GUN=1
S_ACT.PAIR=SDEFAULT.PAIR
S_ACT.RETR=#OPN
S_ACT.CLO_TM=1
S_ACT.PGNO1=43
S_ACT.PGNO2=SDEFAULT.PGNO2
S_ACT.PRESS1=SDEFAULT.PRESS1
S_ACT.PRESS2=SDEFAULT.PRESS2
S_READY=FALSE
PTP Xswp_60_5456
USERSPOT(#SPOT, S_ACT)
WAIT FOR S_READY
;ENDFOLD

;FOLD ; SWP_60_5458;%{PE}%R 8.2.20,%MKUKATPBASIS,%CCOMMENT,%VNORMAL,%P 2:SWP_60_5458
;ENDFOLD
;FOLD PTP swp_60_5458 PDAT26 SPOT Gun=1 RETR OPN PgNo1=44 ACTIVE=1 Tool[2]:Gun C1 Base[1]:Actros;%{PE}%R 8.2.2,%MKUKATPSPOT,%CSPOT,%VPTP,%P 1:PTP, 2:swp_60_5458, 3:, 5:100, 7:PDAT26, 10:1, 12:#FIRST, 14:#OPN, 16:44, 18:1, 20:0, 22:0, 24:1, 25:NORMAL
$BWDSTART=FALSE
PDAT_ACT=PPDAT26
FDAT_ACT=Fswp_60_5458
BAS(#PTP_PARAMS,PPDAT26.VEL)
S_ACT.GUN=1
S_ACT.PAIR=SDEFAULT.PAIR
S_ACT.RETR=#OPN
S_ACT.CLO_TM=1
S_ACT.PGNO1=44
S_ACT.PGNO2=SDEFAULT.PGNO2
S_ACT.PRESS1=SDEFAULT.PRESS1
S_ACT.PRESS2=SDEFAULT.PRESS2
S_READY=FALSE
PTP Xswp_60_5458
USERSPOT(#SPOT, S_ACT)
WAIT FOR S_READY
;ENDFOLD

;FOLD ; SWP_60_5460;%{PE}%R 8.2.20,%MKUKATPBASIS,%CCOMMENT,%VNORMAL,%P 2:SWP_60_5460
;ENDFOLD
;FOLD PTP swp_60_5460 PDAT27 SPOT Gun=1 RETR OPN PgNo1=45 ACTIVE=1 Tool[2]:Gun C1 Base[1]:Actros;%{PE}%R 8.2.2,%MKUKATPSPOT,%CSPOT,%VPTP,%P 1:PTP, 2:swp_60_5460, 3:, 5:100, 7:PDAT27, 10:1, 12:#FIRST, 14:#OPN, 16:45, 18:1, 20:0, 22:0, 24:1, 25:NORMAL
$BWDSTART=FALSE
PDAT_ACT=PPDAT27
FDAT_ACT=Fswp_60_5460
BAS(#PTP_PARAMS,PPDAT27.VEL)
S_ACT.GUN=1
S_ACT.PAIR=SDEFAULT.PAIR
S_ACT.RETR=#OPN
S_ACT.CLO_TM=1
S_ACT.PGNO1=45
S_ACT.PGNO2=SDEFAULT.PGNO2
S_ACT.PRESS1=SDEFAULT.PRESS1
S_ACT.PRESS2=SDEFAULT.PRESS2
S_READY=FALSE
PTP Xswp_60_5460
USERSPOT(#SPOT, S_ACT)
WAIT FOR S_READY
;ENDFOLD

;FOLD ; SWP_60_5462;%{PE}%R 8.2.20,%MKUKATPBASIS,%CCOMMENT,%VNORMAL,%P 2:SWP_60_5462
;ENDFOLD
;FOLD PTP swp_60_5462 PDAT28 SPOT Gun=1 RETR OPN PgNo1=46 ACTIVE=1 Tool[2]:Gun C1 Base[1]:Actros;%{PE}%R 8.2.2,%MKUKATPSPOT,%CSPOT,%VPTP,%P 1:PTP, 2:swp_60_5462, 3:, 5:100, 7:PDAT28, 10:1, 12:#FIRST, 14:#OPN, 16:46, 18:1, 20:0, 22:0, 24:1, 25:NORMAL
$BWDSTART=FALSE
PDAT_ACT=PPDAT28
FDAT_ACT=Fswp_60_5462
BAS(#PTP_PARAMS,PPDAT28.VEL)
S_ACT.GUN=1
S_ACT.PAIR=SDEFAULT.PAIR
S_ACT.RETR=#OPN
S_ACT.CLO_TM=1
S_ACT.PGNO1=46
S_ACT.PGNO2=SDEFAULT.PGNO2
S_ACT.PRESS1=SDEFAULT.PRESS1
S_ACT.PRESS2=SDEFAULT.PRESS2
S_READY=FALSE
PTP Xswp_60_5462
USERSPOT(#SPOT, S_ACT)
WAIT FOR S_READY
;ENDFOLD

;FOLD ; SWP_60_5464;%{PE}%R 8.2.20,%MKUKATPBASIS,%CCOMMENT,%VNORMAL,%P 2:SWP_60_5464
;ENDFOLD
;FOLD PTP swp_60_5464 PDAT29 SPOT Gun=1 RETR OPN PgNo1=47 ACTIVE=1 Tool[2]:Gun C1 Base[1]:Actros;%{PE}%R 8.2.2,%MKUKATPSPOT,%CSPOT,%VPTP,%P 1:PTP, 2:swp_60_5464, 3:, 5:100, 7:PDAT29, 10:1, 12:#FIRST, 14:#OPN, 16:47, 18:1, 20:0, 22:0, 24:1, 25:NORMAL
$BWDSTART=FALSE
PDAT_ACT=PPDAT29
FDAT_ACT=Fswp_60_5464
BAS(#PTP_PARAMS,PPDAT29.VEL)
S_ACT.GUN=1
S_ACT.PAIR=SDEFAULT.PAIR
S_ACT.RETR=#OPN
S_ACT.CLO_TM=1
S_ACT.PGNO1=47
S_ACT.PGNO2=SDEFAULT.PGNO2
S_ACT.PRESS1=SDEFAULT.PRESS1
S_ACT.PRESS2=SDEFAULT.PRESS2
S_READY=FALSE
PTP Xswp_60_5464
USERSPOT(#SPOT, S_ACT)
WAIT FOR S_READY
;ENDFOLD

;FOLD ; SWP_60_5466;%{PE}%R 8.2.20,%MKUKATPBASIS,%CCOMMENT,%VNORMAL,%P 2:SWP_60_5466
;ENDFOLD
;FOLD PTP swp_60_5466 PDAT30 SPOT Gun=1 RETR OPN PgNo1=48 ACTIVE=1 Tool[2]:Gun C1 Base[1]:Actros;%{PE}%R 8.2.2,%MKUKATPSPOT,%CSPOT,%VPTP,%P 1:PTP, 2:swp_60_5466, 3:, 5:100, 7:PDAT30, 10:1, 12:#FIRST, 14:#OPN, 16:48, 18:1, 20:0, 22:0, 24:1, 25:NORMAL
$BWDSTART=FALSE
PDAT_ACT=PPDAT30
FDAT_ACT=Fswp_60_5466
BAS(#PTP_PARAMS,PPDAT30.VEL)
S_ACT.GUN=1
S_ACT.PAIR=SDEFAULT.PAIR
S_ACT.RETR=#OPN
S_ACT.CLO_TM=1
S_ACT.PGNO1=48
S_ACT.PGNO2=SDEFAULT.PGNO2
S_ACT.PRESS1=SDEFAULT.PRESS1
S_ACT.PRESS2=SDEFAULT.PRESS2
S_READY=FALSE
PTP Xswp_60_5466
USERSPOT(#SPOT, S_ACT)
WAIT FOR S_READY
;ENDFOLD

;FOLD ; SWP_60_5468;%{PE}%R 8.2.20,%MKUKATPBASIS,%CCOMMENT,%VNORMAL,%P 2:SWP_60_5468
;ENDFOLD
;FOLD PTP swp_60_5468 PDAT31 SPOT Gun=1 RETR OPN PgNo1=49 ACTIVE=1 Tool[2]:Gun C1 Base[1]:Actros;%{PE}%R 8.2.2,%MKUKATPSPOT,%CSPOT,%VPTP,%P 1:PTP, 2:swp_60_5468, 3:, 5:100, 7:PDAT31, 10:1, 12:#FIRST, 14:#OPN, 16:49, 18:1, 20:0, 22:0, 24:1, 25:NORMAL
$BWDSTART=FALSE
PDAT_ACT=PPDAT31
FDAT_ACT=Fswp_60_5468
BAS(#PTP_PARAMS,PPDAT31.VEL)
S_ACT.GUN=1
S_ACT.PAIR=SDEFAULT.PAIR
S_ACT.RETR=#OPN
S_ACT.CLO_TM=1
S_ACT.PGNO1=49
S_ACT.PGNO2=SDEFAULT.PGNO2
S_ACT.PRESS1=SDEFAULT.PRESS1
S_ACT.PRESS2=SDEFAULT.PRESS2
S_READY=FALSE
PTP Xswp_60_5468
USERSPOT(#SPOT, S_ACT)
WAIT FOR S_READY
;ENDFOLD

;FOLD ; SWP_60_5470;%{PE}%R 8.2.20,%MKUKATPBASIS,%CCOMMENT,%VNORMAL,%P 2:SWP_60_5470
;ENDFOLD
;FOLD PTP swp_60_5470 PDAT32 SPOT Gun=1 RETR OPN PgNo1=50 ACTIVE=1 Tool[2]:Gun C1 Base[1]:Actros;%{PE}%R 8.2.2,%MKUKATPSPOT,%CSPOT,%VPTP,%P 1:PTP, 2:swp_60_5470, 3:, 5:100, 7:PDAT32, 10:1, 12:#FIRST, 14:#OPN, 16:50, 18:1, 20:0, 22:0, 24:1, 25:NORMAL
$BWDSTART=FALSE
PDAT_ACT=PPDAT32
FDAT_ACT=Fswp_60_5470
BAS(#PTP_PARAMS,PPDAT32.VEL)
S_ACT.GUN=1
S_ACT.PAIR=SDEFAULT.PAIR
S_ACT.RETR=#OPN
S_ACT.CLO_TM=1
S_ACT.PGNO1=50
S_ACT.PGNO2=SDEFAULT.PGNO2
S_ACT.PRESS1=SDEFAULT.PRESS1
S_ACT.PRESS2=SDEFAULT.PRESS2
S_READY=FALSE
PTP Xswp_60_5470
USERSPOT(#SPOT, S_ACT)
WAIT FOR S_READY
;ENDFOLD

;FOLD ; SWP_60_5472;%{PE}%R 8.2.20,%MKUKATPBASIS,%CCOMMENT,%VNORMAL,%P 2:SWP_60_5472
;ENDFOLD
;FOLD PTP swp_60_5472 PDAT33 SPOT Gun=1 RETR OPN PgNo1=51 ACTIVE=1 Tool[2]:Gun C1 Base[1]:Actros;%{PE}%R 8.2.2,%MKUKATPSPOT,%CSPOT,%VPTP,%P 1:PTP, 2:swp_60_5472, 3:, 5:100, 7:PDAT33, 10:1, 12:#FIRST, 14:#OPN, 16:51, 18:1, 20:0, 22:0, 24:1, 25:NORMAL
$BWDSTART=FALSE
PDAT_ACT=PPDAT33
FDAT_ACT=Fswp_60_5472
BAS(#PTP_PARAMS,PPDAT33.VEL)
S_ACT.GUN=1
S_ACT.PAIR=SDEFAULT.PAIR
S_ACT.RETR=#OPN
S_ACT.CLO_TM=1
S_ACT.PGNO1=51
S_ACT.PGNO2=SDEFAULT.PGNO2
S_ACT.PRESS1=SDEFAULT.PRESS1
S_ACT.PRESS2=SDEFAULT.PRESS2
S_READY=FALSE
PTP Xswp_60_5472
USERSPOT(#SPOT, S_ACT)
WAIT FOR S_READY
;ENDFOLD

;FOLD PTP P8 CONT Vel=100 % PDAT59 Tool[2]:Gun C1 Base[1]:Actros;%{PE}%R 8.2.20,%MKUKATPBASIS,%CMOVE,%VPTP,%P 1:PTP, 2:P8, 3:C_DIS, 5:100, 7:PDAT59
$BWDSTART=FALSE
PDAT_ACT=PPDAT59
FDAT_ACT=FP8
BAS(#PTP_PARAMS,100)
PTP XP8 C_DIS
;ENDFOLD

;FOLD ; SWP_60_5474;%{PE}%R 8.2.20,%MKUKATPBASIS,%CCOMMENT,%VNORMAL,%P 2:SWP_60_5474
;ENDFOLD
;FOLD PTP swp_60_5474 PDAT34 SPOT Gun=1 RETR OPN PgNo1=52 ACTIVE=1 Tool[2]:Gun C1 Base[1]:Actros;%{PE}%R 8.2.2,%MKUKATPSPOT,%CSPOT,%VPTP,%P 1:PTP, 2:swp_60_5474, 3:, 5:100, 7:PDAT34, 10:1, 12:#FIRST, 14:#OPN, 16:52, 18:1, 20:0, 22:0, 24:1, 25:NORMAL
$BWDSTART=FALSE
PDAT_ACT=PPDAT34
FDAT_ACT=Fswp_60_5474
BAS(#PTP_PARAMS,PPDAT34.VEL)
S_ACT.GUN=1
S_ACT.PAIR=SDEFAULT.PAIR
S_ACT.RETR=#OPN
S_ACT.CLO_TM=1
S_ACT.PGNO1=52
S_ACT.PGNO2=SDEFAULT.PGNO2
S_ACT.PRESS1=SDEFAULT.PRESS1
S_ACT.PRESS2=SDEFAULT.PRESS2
S_READY=FALSE
PTP Xswp_60_5474
USERSPOT(#SPOT, S_ACT)
WAIT FOR S_READY
;ENDFOLD

;FOLD ; SWP_60_5476;%{PE}%R 8.2.20,%MKUKATPBASIS,%CCOMMENT,%VNORMAL,%P 2:SWP_60_5476
;ENDFOLD
;FOLD PTP swp_60_5476 PDAT35 SPOT Gun=1 RETR OPN PgNo1=53 ACTIVE=1 Tool[2]:Gun C1 Base[1]:Actros;%{PE}%R 8.2.2,%MKUKATPSPOT,%CSPOT,%VPTP,%P 1:PTP, 2:swp_60_5476, 3:, 5:100, 7:PDAT35, 10:1, 12:#FIRST, 14:#OPN, 16:53, 18:1, 20:0, 22:0, 24:1, 25:NORMAL
$BWDSTART=FALSE
PDAT_ACT=PPDAT35
FDAT_ACT=Fswp_60_5476
BAS(#PTP_PARAMS,PPDAT35.VEL)
S_ACT.GUN=1
S_ACT.PAIR=SDEFAULT.PAIR
S_ACT.RETR=#OPN
S_ACT.CLO_TM=1
S_ACT.PGNO1=53
S_ACT.PGNO2=SDEFAULT.PGNO2
S_ACT.PRESS1=SDEFAULT.PRESS1
S_ACT.PRESS2=SDEFAULT.PRESS2
S_READY=FALSE
PTP Xswp_60_5476
USERSPOT(#SPOT, S_ACT)
WAIT FOR S_READY
;ENDFOLD

;FOLD PTP p43 CONT Vel=100 % P_OLP51 Tool[2]:Gun C1 Base[1]:Actros;%{PE}%R 8.2.20,%MKUKATPBASIS,%CMOVE,%VPTP,%P 1:PTP, 2:p43, 3:C_DIS, 5:100, 7:P_OLP51
$BWDSTART=FALSE
PDAT_ACT=PP_OLP51
FDAT_ACT=Fp43
BAS(#PTP_PARAMS,100)
PTP Xp43 C_DIS
;ENDFOLD
;FOLD PTP p44 CONT Vel=100 % P_OLP52 Tool[2]:Gun C1 Base[1]:Actros;%{PE}%R8.2,%MKUKATPBASIS,%CMOVE,%VPTP,%P 1:PTP, 2:p44, 3:C_DIS, 5:100, 7:P_OLP52
$BWDSTART = FALSE
PDAT_ACT= PP_OLP52
FDAT_ACT= Fp44
BAS(#PTP_PARAMS,100)
PTP Xp44 C_DIS
;ENDFOLD

;FOLD OUT 3339 'R5 SOLDANDO' State=FALSE ;%{PE}%R 8.2.20,%MKUKATPBASIS,%COUT,%VOUTX,%P 2:3339, 3:R5 SOLDANDO, 5:FALSE, 6:
$OUT[3339]=FALSE
;ENDFOLD
;FOLD OUT 3340 'locking-signal PLC' State=TRUE ;%{PE}%R 8.2.20,%MKUKATPBASIS,%COUT,%VOUTX,%P 2:3340, 3:locking-signal PLC, 5:TRUE, 6:
$OUT[3340]=TRUE
;ENDFOLD

;FOLD LIN p45 CONT Vel=2 m/s CPDAT1 Tool[2]:Gun C1 Base[1]:Actros;%{PE}%R 8.2.20,%MKUKATPBASIS,%CMOVE,%VLIN,%P 1:LIN, 2:p45, 3:C_DIS C_DIS, 5:2, 7:CPDAT1
$BWDSTART=FALSE
LDAT_ACT=LCPDAT1
FDAT_ACT=Fp45
BAS(#CP_PARAMS,2)
LIN Xp45 C_DIS C_DIS
;ENDFOLD

;FOLD PTP P5 Vel=100 % PDAT56 Tool[2]:Gun C1 Base[1]:Actros;%{PE}%R 8.2.20,%MKUKATPBASIS,%CMOVE,%VPTP,%P 1:PTP, 2:P5, 3:, 5:100, 7:PDAT56
$BWDSTART=FALSE
PDAT_ACT=PPDAT56
FDAT_ACT=FP5
BAS(#PTP_PARAMS,100)
PTP XP5
;ENDFOLD

IF(NOT(GHOST())) THEN
IF FraesAnf (1) THEN

;FOLD PTP pFresa_01 CONT Vel=100 % PDAT44 Tool[2]:Gun C1 Base[1]:Actros;%{PE}%R 8.2.20,%MKUKATPBASIS,%CMOVE,%VPTP,%P 1:PTP, 2:pFresa_01, 3:C_DIS, 5:100, 7:PDAT44
$BWDSTART=FALSE
PDAT_ACT=PPDAT44
FDAT_ACT=FpFresa_01
BAS(#PTP_PARAMS,100)
PTP XpFresa_01 C_DIS
;ENDFOLD
;FOLD PULSE 168 'DOCK 1 Fechar Proteção' State=TRUE Time=1 sec;%{PE}%R 8.2.20,%MKUKATPBASIS,%COUT,%VPULSE,%P 2:168, 3:DOCK 1 Fechar Proteção, 5:TRUE, 6:, 8:1
PULSE($OUT[168], TRUE,1)
;ENDFOLD
;FOLD WAIT FOR ( IN 166 'DOCK 1 Proteção Fechada' );%{PE}%R 8.2.20,%MKUKATPBASIS,%CEXT_WAIT_FOR,%VEXT_WAIT_FOR,%P 2:, 4:, 5:$IN, 6:166, 7:DOCK 1 Proteção Fechada, 9:
WAIT FOR  ( $IN[166] )
;ENDFOLD
;FOLD PTP pFresa_02 CONT Vel=100 % PDAT45 Tool[2]:Gun C1 Base[1]:Actros;%{PE}%R 8.2.20,%MKUKATPBASIS,%CMOVE,%VPTP,%P 1:PTP, 2:pFresa_02, 3:C_DIS, 5:100, 7:PDAT45
$BWDSTART=FALSE
PDAT_ACT=PPDAT45
FDAT_ACT=FpFresa_02
BAS(#PTP_PARAMS,100)
PTP XpFresa_02 C_DIS
;ENDFOLD
 f_Fraes_2()
;FOLD PTP pFresa_03 CONT Vel=100 % PDAT46 Tool[2]:Gun C1 Base[1]:Actros;%{PE}%R 8.2.20,%MKUKATPBASIS,%CMOVE,%VPTP,%P 1:PTP, 2:pFresa_03, 3:C_DIS, 5:100, 7:PDAT46
$BWDSTART=FALSE
PDAT_ACT=PPDAT46
FDAT_ACT=FpFresa_03
BAS(#PTP_PARAMS,100)
PTP XpFresa_03 C_DIS
;ENDFOLD
;FOLD PTP pFresa_04 CONT Vel=100 % PDAT47 Tool[2]:Gun C1 Base[1]:Actros;%{PE}%R 8.2.20,%MKUKATPBASIS,%CMOVE,%VPTP,%P 1:PTP, 2:pFresa_04, 3:C_DIS, 5:100, 7:PDAT47
$BWDSTART=FALSE
PDAT_ACT=PPDAT47
FDAT_ACT=FpFresa_04
BAS(#PTP_PARAMS,100)
PTP XpFresa_04 C_DIS
;ENDFOLD
ENDIF
ENDIF
;FOLD PTP P6 Vel=100 % PDAT57 Tool[2]:Gun C1 Base[1]:Actros;%{PE}%R 8.2.20,%MKUKATPBASIS,%CMOVE,%VPTP,%P 1:PTP, 2:P6, 3:, 5:100, 7:PDAT57
$BWDSTART=FALSE
PDAT_ACT=PPDAT57
FDAT_ACT=FP6
BAS(#PTP_PARAMS,100)
PTP XP6
;ENDFOLD
;FOLD PTP P7 Vel=100 % PDAT58 Tool[2]:Gun C1 Base[1]:Actros;%{PE}%R 8.2.20,%MKUKATPBASIS,%CMOVE,%VPTP,%P 1:PTP, 2:P7, 3:, 5:100, 7:PDAT58
$BWDSTART=FALSE
PDAT_ACT=PPDAT58
FDAT_ACT=FP7
BAS(#PTP_PARAMS,100)
PTP XP7
;ENDFOLD

IF ($IN[3342]) OR ($IN[3341]) THEN
ENDIF

;FOLD OUT 3339 'R5 SOLDANDO' State=TRUE CONT;%{PE}%R 8.2.20,%MKUKATPBASIS,%COUT,%VOUTX,%P 2:3339, 3:R5 SOLDANDO, 5:TRUE, 6:CONTINUE
CONTINUE
$OUT[3339]=TRUE
;ENDFOLD
END

--- ps_r5_l_resp1_c1_mod.dat ---
&ACCESS RVO1
&REL 40
&COMMENT C1 Respot LTA/LTB/MGS/MGSB
&PARAM DISKPATH = KRC:\R1\Program\SOLDA LTC
DEFDAT  ps_r5_l_resp1_c1_mod
;FOLD EXTERNAL DECLARATIONS;%{PE}%MKUKATPBASIS,%CEXT,%VCOMMON,%P
;FOLD GRIPPERTECH EXT
EXT  H50 (INT  :IN,INT  :IN,INT  :IN,GRP_TYP  :IN )
;ENDFOLD (GRIPPERTECH EXT)
;FOLD SPOTTECH EXT
EXT  USERSPOT (S_COMMAND  :IN,SPOT_TYPE  :IN )
;ENDFOLD (SPOTTECH EXT)
;FOLD BASISTECH EXT;%{PE}%MKUKATPBASIS,%CEXT,%VEXT,%P
EXT  BAS (BAS_COMMAND  :IN,REAL  :IN )
DECL INT SUCCESS
;ENDFOLD (BASISTECH EXT)
;FOLD USER EXT;%{E}%MKUKATPUSER,%CEXT,%VEXT,%P
;Make your modifications here

;ENDFOLD (USER EXT)
;ENDFOLD (EXTERNAL DECLARATIONS)

;# ============ START PATH : swp_p13060r5_l_resp1_c1 =============
DECL FDAT Fp27={TOOL_NO 2,BASE_NO 1,IPO_FRAME #BASE,POINT2[] " "}
DECL PDAT PP_OLP2={VEL 100.0,ACC 100.0,APO_DIST 100.0,APO_MODE #CDIS}
DECL E6POS Xp27={X 1845.81897,Y -593.418579,Z 1603.97095,A -121.989098,B 59.1542511,C 72.0093231,S 2,T 11,E1 0.0,E2 0.0,E3 0.0,E4 0.0,E5 0.0,E6 0.0}
DECL FDAT Fp28={TOOL_NO 2,BASE_NO 1,IPO_FRAME #BASE,POINT2[] " ",TQ_STATE FALSE}
DECL PDAT PP_OLP3={VEL 100.0,ACC 100.0,APO_DIST 100.0,APO_MODE #CDIS}
DECL E6POS Xp28={X 1997.50305,Y -891.716003,Z 484.907013,A -90.0,B 70.0,C 90.0,S 2,T 9}
DECL FDAT Fp29={TOOL_NO 2,BASE_NO 1,IPO_FRAME #BASE,POINT2[] " "}
DECL PDAT PP_OLP4={VEL 100.0,ACC 100.0,APO_DIST 100.0,APO_MODE #CDIS}
DECL E6POS Xp29={X 2139.23706,Y -917.971313,Z 485.162598,A -90.0011368,B 55.4054489,C 89.9988022,S 2,T 9,E1 0.0,E2 0.0,E3 0.0,E4 0.0,E5 0.0,E6 0.0}
DECL FDAT Fswp_60_5475={TOOL_NO 2,BASE_NO 1,IPO_FRAME #BASE,POINT2[] " ",TQ_STATE FALSE}
DECL SPOT_TYPE SS_OLP1={GUN 2,PAIR #FIRST,RETR #CLO,CLO_TM 0,PGNO1 1,PRESS1 1.0,PGNO2 0,PRESS2 0.0}
DECL E6POS Xswp_60_5475={X 2135.90894,Y -911.47467,Z 453.372406,A -89.9971771,B 55.4051208,C 90.0001526,S 2,T 9,E1 0.0,E2 0.0,E3 0.0,E4 0.0,E5 0.0,E6 0.0}
DECL FDAT Fp30={TOOL_NO 2,BASE_NO 1,IPO_FRAME #BASE,POINT2[] " "}
DECL PDAT PP_OLP6={VEL 100.0,ACC 100.0,APO_DIST 100.0,APO_MODE #CDIS}
DECL E6POS Xp30={X 2131.08301,Y -852.001526,Z 555.870117,A -89.4855194,B 67.1472626,C 90.4478836,S 2,T 9,E1 0.0,E2 0.0,E3 0.0,E4 0.0,E5 0.0,E6 0.0}
DECL FDAT Fp31={TOOL_NO 2,BASE_NO 1,IPO_FRAME #BASE,POINT2[] " "}
DECL PDAT PP_OLP7={VEL 100.0,ACC 100.0,APO_DIST 100.0,APO_MODE #CDIS}
DECL E6POS Xp31={X 2137.42505,Y -722.042297,Z 489.846588,A -88.7272797,B 81.037262,C 91.257431,S 2,T 9,E1 0.0,E2 0.0,E3 0.0,E4 0.0,E5 0.0,E6 0.0}
DECL FDAT Fswp_60_5469={TOOL_NO 2,BASE_NO 1,IPO_FRAME #BASE,POINT2[] " "}
DECL SPOT_TYPE SS_OLP2={GUN 1,PAIR #FIRST,RETR #CLO,CLO_TM 0,PGNO1 1,PRESS1 1.0,PGNO2 0,PRESS2 0.0}
DECL E6POS Xswp_60_5469={X 2131.29492,Y -717.034912,Z 453.877014,A -90.021492,B 82.3450699,C 89.9891205,S 2,T 9,E1 0.0,E2 0.0,E3 0.0,E4 0.0,E5 0.0,E6 0.0}
DECL FDAT Fswp_60_5467={TOOL_NO 2,BASE_NO 1,IPO_FRAME #BASE,POINT2[] " "}
DECL SPOT_TYPE SS_OLP3={GUN 2,PAIR #FIRST,RETR #CLO,CLO_TM 0,PGNO1 1,PRESS1 1.0,PGNO2 0,PRESS2 0.0}
DECL E6POS Xswp_60_5467={X 2133.63892,Y -684.341125,Z 452.95871,A -89.9840393,B 82.3411789,C 90.0279465,S 2,T 9,E1 0.0,E2 0.0,E3 0.0,E4 0.0,E5 0.0,E6 0.0}
DECL FDAT Fswp_60_5465={TOOL_NO 2,BASE_NO 1,IPO_FRAME #BASE,POINT2[] " "}
DECL SPOT_TYPE SS_OLP4={GUN 2,PAIR #FIRST,RETR #CLO,CLO_TM 0,PGNO1 1,PRESS1 1.0,PGNO2 0,PRESS2 0.0}
DECL E6POS Xswp_60_5465={X 2132.70093,Y -642.964417,Z 455.538086,A -90.0013123,B 82.3429031,C 90.0109177,S 2,T 9,E1 0.0,E2 0.0,E3 0.0,E4 0.0,E5 0.0,E6 0.0}
DECL FDAT Fswp_60_5463={TOOL_NO 2,BASE_NO 1,IPO_FRAME #BASE,POINT2[] " "}
DECL SPOT_TYPE SS_OLP5={GUN 2,PAIR #FIRST,RETR #CLO,CLO_TM 0,PGNO1 1,PRESS1 1.0,PGNO2 0,PRESS2 0.0}
DECL E6POS Xswp_60_5463={X 2133.63403,Y -595.48291,Z 459.121307,A -90.0429077,B 82.338707,C 89.9643173,S 2,T 9,E1 0.0,E2 0.0,E3 0.0,E4 0.0,E5 0.0,E6 0.0}
DECL FDAT Fswp_60_5461={TOOL_NO 2,BASE_NO 1,IPO_FRAME #BASE,POINT2[] " "}
DECL SPOT_TYPE SS_OLP6={GUN 2,PAIR #FIRST,RETR #CLO,CLO_TM 0,PGNO1 1,PRESS1 1.0,PGNO2 0,PRESS2 0.0}
DECL E6POS Xswp_60_5461={X 2131.61304,Y -545.615173,Z 458.831085,A -89.9837799,B 82.3423767,C 90.0268021,S 2,T 9,E1 0.0,E2 0.0,E3 0.0,E4 0.0,E5 0.0,E6 0.0}
DECL FDAT Fswp_60_5459={TOOL_NO 2,BASE_NO 1,IPO_FRAME #BASE,POINT2[] " "}
DECL SPOT_TYPE SS_OLP7={GUN 2,PAIR #FIRST,RETR #CLO,CLO_TM 0,PGNO1 1,PRESS1 1.0,PGNO2 0,PRESS2 0.0}
DECL E6POS Xswp_60_5459={X 2132.04102,Y -495.496887,Z 458.613007,A -89.9970169,B 82.3421936,C 90.0136337,S 2,T 9,E1 0.0,E2 0.0,E3 0.0,E4 0.0,E5 0.0,E6 0.0}
DECL FDAT Fswp_60_5457={TOOL_NO 2,BASE_NO 1,IPO_FRAME #BASE,POINT2[] " "}
DECL SPOT_TYPE SS_OLP8={GUN 2,PAIR #FIRST,RETR #CLO,CLO_TM 0,PGNO1 1,PRESS1 1.0,PGNO2 0,PRESS2 0.0}
DECL E6POS Xswp_60_5457={X 2130.80591,Y -445.484497,Z 458.331207,A -89.9970169,B 82.3421936,C 90.0136337,S 2,T 9,E1 0.0,E2 0.0,E3 0.0,E4 0.0,E5 0.0,E6 0.0}
DECL FDAT Fswp_60_5455={TOOL_NO 2,BASE_NO 1,IPO_FRAME #BASE,POINT2[] " "}
DECL SPOT_TYPE SS_OLP9={GUN 2,PAIR #FIRST,RETR #CLO,CLO_TM 0,PGNO1 1,PRESS1 1.0,PGNO2 0,PRESS2 0.0}
DECL E6POS Xswp_60_5455={X 2130.73511,Y -395.919586,Z 458.193604,A -89.9978638,B 82.3421631,C 90.0126801,S 2,T 9,E1 0.0,E2 0.0,E3 0.0,E4 0.0,E5 0.0,E6 0.0}
DECL FDAT Fswp_60_5453={TOOL_NO 2,BASE_NO 1,IPO_FRAME #BASE,POINT2[] " ",TQ_STATE FALSE}
DECL SPOT_TYPE SS_OLP10={GUN 2,PAIR #FIRST,RETR #CLO,CLO_TM 0,PGNO1 1,PRESS1 1.0,PGNO2 0,PRESS2 0.0}
DECL E6POS Xswp_60_5453={X 2131.04297,Y -345.1315,Z 457.56781,A -89.9977875,B 82.3409729,C 90.0127563,S 2,T 9,E1 0.0,E2 0.0,E3 0.0,E4 0.0,E5 0.0,E6 0.0}
DECL FDAT Fswp_60_5451={TOOL_NO 2,BASE_NO 1,IPO_FRAME #BASE,POINT2[] " "}
DECL SPOT_TYPE SS_OLP11={GUN 2,PAIR #FIRST,RETR #CLO,CLO_TM 0,PGNO1 1,PRESS1 1.0,PGNO2 0,PRESS2 0.0}
DECL E6POS Xswp_60_5451={X 2129.9231,Y -294.872101,Z 458.254486,A -90.0284195,B 82.342453,C 90.0143509,S 2,T 9,E1 0.0,E2 0.0,E3 0.0,E4 0.0,E5 0.0,E6 0.0}
DECL FDAT Fswp_60_5449={TOOL_NO 2,BASE_NO 1,IPO_FRAME #BASE,POINT2[] " "}
DECL SPOT_TYPE SS_OLP12={GUN 2,PAIR #FIRST,RETR #CLO,CLO_TM 0,PGNO1 1,PRESS1 1.0,PGNO2 0,PRESS2 0.0}
DECL E6POS Xswp_60_5449={X 2128.29297,Y -244.150894,Z 458.978485,A -90.0126572,B 82.3440018,C 90.0295868,S 2,T 9,E1 0.0,E2 0.0,E3 0.0,E4 0.0,E5 0.0,E6 0.0}
DECL FDAT Fswp_60_5447={TOOL_NO 2,BASE_NO 1,IPO_FRAME #BASE,POINT2[] " "}
DECL SPOT_TYPE SS_OLP13={GUN 2,PAIR #FIRST,RETR #CLO,CLO_TM 0,PGNO1 1,PRESS1 1.0,PGNO2 0,PRESS2 0.0}
DECL E6POS Xswp_60_5447={X 2129.25195,Y -196.220306,Z 457.147888,A -90.0221176,B 82.3441162,C 90.02034,S 2,T 9,E1 0.0,E2 0.0,E3 0.0,E4 0.0,E5 0.0,E6 0.0}
DECL FDAT Fswp_60_5445={TOOL_NO 2,BASE_NO 1,IPO_FRAME #BASE,POINT2[] " "}
DECL SPOT_TYPE SS_OLP14={GUN 2,PAIR #FIRST,RETR #CLO,CLO_TM 0,PGNO1 1,PRESS1 1.0,PGNO2 0,PRESS2 0.0}
DECL E6POS Xswp_60_5445={X 2128.21899,Y -145.126602,Z 457.275787,A -90.0608368,B 82.6251526,C 89.9777069,S 2,T 9,E1 0.0,E2 0.0,E3 0.0,E4 0.0,E5 0.0,E6 0.0}
DECL FDAT Fswp_60_5443={TOOL_NO 2,BASE_NO 1,IPO_FRAME #BASE,POINT2[] " "}
DECL SPOT_TYPE SS_OLP15={GUN 2,PAIR #FIRST,RETR #CLO,CLO_TM 0,PGNO1 1,PRESS1 1.0,PGNO2 0,PRESS2 0.0}
DECL E6POS Xswp_60_5443={X 2127.63599,Y -95.1643677,Z 456.787994,A -90.0564728,B 82.6244431,C 89.9812164,S 2,T 9,E1 0.0,E2 0.0,E3 0.0,E4 0.0,E5 0.0,E6 0.0}
DECL SPOT_TYPE SS_OLP16={GUN 2,PAIR #FIRST,RETR #CLO,CLO_TM 0,PGNO1 1,PRESS1 1.0,PGNO2 0,PRESS2 0.0}
DECL FDAT Fswp_60_5442={TOOL_NO 2,BASE_NO 1,IPO_FRAME #BASE,POINT2[] " ",TQ_STATE FALSE}
DECL SPOT_TYPE SS_OLP17={GUN 2,PAIR #FIRST,RETR #CLO,CLO_TM 0,PGNO1 1,PRESS1 1.0,PGNO2 0,PRESS2 0.0}
DECL E6POS Xswp_60_5442={X 2126.58594,Y 64.7783432,Z 457.138885,A -89.7387772,B 71.7323685,C 90.6889038,S 2,T 8,E1 0.0,E2 0.0,E3 0.0,E4 0.0,E5 0.0,E6 0.0}
DECL FDAT Fswp_60_5444={TOOL_NO 2,BASE_NO 1,IPO_FRAME #BASE,POINT2[] " "}
DECL SPOT_TYPE SS_OLP18={GUN 2,PAIR #FIRST,RETR #CLO,CLO_TM 0,PGNO1 1,PRESS1 1.0,PGNO2 0,PRESS2 0.0}
DECL E6POS Xswp_60_5444={X 2126.28101,Y 103.0009,Z 455.710205,A -90.0737915,B 82.6281433,C 89.9679184,S 2,T 0,E1 0.0,E2 0.0,E3 0.0,E4 0.0,E5 0.0,E6 0.0}
DECL FDAT Fswp_60_5446={TOOL_NO 2,BASE_NO 1,IPO_FRAME #BASE,POINT2[] " "}
DECL SPOT_TYPE SS_OLP19={GUN 2,PAIR #FIRST,RETR #CLO,CLO_TM 0,PGNO1 1,PRESS1 1.0,PGNO2 0,PRESS2 0.0}
DECL E6POS Xswp_60_5446={X 2122.77905,Y 143.274506,Z 455.516602,A -89.2510529,B 89.9936905,C 90.7095032,S 2,T 0,E1 0.0,E2 0.0,E3 0.0,E4 0.0,E5 0.0,E6 0.0}
DECL FDAT Fswp_60_5448={TOOL_NO 2,BASE_NO 1,IPO_FRAME #BASE,POINT2[] " "}
DECL SPOT_TYPE SS_OLP20={GUN 2,PAIR #FIRST,RETR #CLO,CLO_TM 0,PGNO1 1,PRESS1 1.0,PGNO2 0,PRESS2 0.0}
DECL E6POS Xswp_60_5448={X 2122.31494,Y 196.526993,Z 456.286804,A -101.823601,B 89.9973907,C 78.1410065,S 2,T 0,E1 0.0,E2 0.0,E3 0.0,E4 0.0,E5 0.0,E6 0.0}
DECL FDAT Fswp_60_5450={TOOL_NO 2,BASE_NO 1,IPO_FRAME #BASE,POINT2[] " "}
DECL SPOT_TYPE SS_OLP21={GUN 2,PAIR #FIRST,RETR #CLO,CLO_TM 0,PGNO1 1,PRESS1 1.0,PGNO2 0,PRESS2 0.0}
DECL E6POS Xswp_60_5450={X 2121.8689,Y 254.108994,Z 456.187286,A -94.3674927,B 89.9969177,C 85.5966568,S 2,T 0,E1 0.0,E2 0.0,E3 0.0,E4 0.0,E5 0.0,E6 0.0}
DECL FDAT Fswp_60_5454={TOOL_NO 2,BASE_NO 1,IPO_FRAME #BASE,POINT2[] " "}
DECL SPOT_TYPE SS_OLP22={GUN 2,PAIR #FIRST,RETR #CLO,CLO_TM 0,PGNO1 1,PRESS1 1.0,PGNO2 0,PRESS2 0.0}
DECL E6POS Xswp_60_5454={X 2120.66406,Y 376.444397,Z 455.370087,A -1.18336701,B 89.9984818,C 178.781494,S 2,T 0,E1 0.0,E2 0.0,E3 0.0,E4 0.0,E5 0.0,E6 0.0}
DECL FDAT Fswp_60_5456={TOOL_NO 2,BASE_NO 1,IPO_FRAME #BASE,POINT2[] " "}
DECL SPOT_TYPE SS_OLP23={GUN 2,PAIR #FIRST,RETR #CLO,CLO_TM 0,PGNO1 1,PRESS1 1.0,PGNO2 0,PRESS2 0.0}
DECL E6POS Xswp_60_5456={X 2120.68896,Y 412.821991,Z 454.822601,A -68.3707886,B 89.9970932,C 111.590797,S 2,T 0,E1 0.0,E2 0.0,E3 0.0,E4 0.0,E5 0.0,E6 0.0}
DECL FDAT Fswp_60_5458={TOOL_NO 2,BASE_NO 1,IPO_FRAME #BASE,POINT2[] " "}
DECL SPOT_TYPE SS_OLP24={GUN 2,PAIR #FIRST,RETR #CLO,CLO_TM 0,PGNO1 1,PRESS1 1.0,PGNO2 0,PRESS2 0.0}
DECL E6POS Xswp_60_5458={X 2119.74707,Y 455.093109,Z 455.775909,A 86.7909012,B 89.9962463,C -93.2465363,S 2,T 0,E1 0.0,E2 0.0,E3 0.0,E4 0.0,E5 0.0,E6 0.0}
DECL FDAT Fswp_60_5460={TOOL_NO 2,BASE_NO 1,IPO_FRAME #BASE,POINT2[] " "}
DECL SPOT_TYPE SS_OLP25={GUN 2,PAIR #FIRST,RETR #CLO,CLO_TM 0,PGNO1 1,PRESS1 1.0,PGNO2 0,PRESS2 0.0}
DECL E6POS Xswp_60_5460={X 2117.61694,Y 504.404602,Z 455.413696,A -86.3393631,B 89.9969864,C 93.6218338,S 2,T 0,E1 0.0,E2 0.0,E3 0.0,E4 0.0,E5 0.0,E6 0.0}
DECL FDAT Fswp_60_5462={TOOL_NO 2,BASE_NO 1,IPO_FRAME #BASE,POINT2[] " "}
DECL SPOT_TYPE SS_OLP26={GUN 2,PAIR #FIRST,RETR #CLO,CLO_TM 0,PGNO1 1,PRESS1 1.0,PGNO2 0,PRESS2 0.0}
DECL E6POS Xswp_60_5462={X 2118.40405,Y 558.515076,Z 455.445099,A -94.5428238,B 89.9965363,C 85.4143906,S 2,T 0,E1 0.0,E2 0.0,E3 0.0,E4 0.0,E5 0.0,E6 0.0}
DECL FDAT Fswp_60_5464={TOOL_NO 2,BASE_NO 1,IPO_FRAME #BASE,POINT2[] " "}
DECL SPOT_TYPE SS_OLP27={GUN 2,PAIR #FIRST,RETR #CLO,CLO_TM 0,PGNO1 1,PRESS1 1.0,PGNO2 0,PRESS2 0.0}
DECL E6POS Xswp_60_5464={X 2115.68799,Y 605.4953,Z 455.568787,A -85.6590805,B 89.9949112,C 94.2989273,S 2,T 0,E1 0.0,E2 0.0,E3 0.0,E4 0.0,E5 0.0,E6 0.0}
DECL FDAT Fswp_60_5466={TOOL_NO 2,BASE_NO 1,IPO_FRAME #BASE,POINT2[] " "}
DECL SPOT_TYPE SS_OLP28={GUN 2,PAIR #FIRST,RETR #CLO,CLO_TM 0,PGNO1 1,PRESS1 1.0,PGNO2 0,PRESS2 0.0}
DECL E6POS Xswp_60_5466={X 2115.07007,Y 655.125122,Z 456.385803,A -81.9263535,B 89.9906235,C 98.0294113,S 2,T 0,E1 0.0,E2 0.0,E3 0.0,E4 0.0,E5 0.0,E6 0.0}
DECL FDAT Fswp_60_5468={TOOL_NO 2,BASE_NO 1,IPO_FRAME #BASE,POINT2[] " "}
DECL SPOT_TYPE SS_OLP29={GUN 2,PAIR #FIRST,RETR #CLO,CLO_TM 0,PGNO1 1,PRESS1 1.0,PGNO2 0,PRESS2 0.0}
DECL E6POS Xswp_60_5468={X 2115.62402,Y 704.131287,Z 455.789795,A -34.6977997,B 89.9885025,C 145.260895,S 2,T 0,E1 0.0,E2 0.0,E3 0.0,E4 0.0,E5 0.0,E6 0.0}
DECL FDAT Fswp_60_5470={TOOL_NO 2,BASE_NO 1,IPO_FRAME #BASE,POINT2[] " "}
DECL SPOT_TYPE SS_OLP30={GUN 2,PAIR #FIRST,RETR #CLO,CLO_TM 0,PGNO1 1,PRESS1 1.0,PGNO2 0,PRESS2 0.0}
DECL E6POS Xswp_60_5470={X 2113.56909,Y 751.380981,Z 455.6922,A -132.501495,B 89.9970627,C 47.4606705,S 2,T 0,E1 0.0,E2 0.0,E3 0.0,E4 0.0,E5 0.0,E6 0.0}
DECL FDAT Fswp_60_5472={TOOL_NO 2,BASE_NO 1,IPO_FRAME #BASE,POINT2[] " "}
DECL SPOT_TYPE SS_OLP31={GUN 2,PAIR #FIRST,RETR #CLO,CLO_TM 0,PGNO1 1,PRESS1 1.0,PGNO2 0,PRESS2 0.0}
DECL E6POS Xswp_60_5472={X 2113.7041,Y 802.497986,Z 456.029297,A 90.4704666,B 89.5185623,C -89.5709686,S 2,T 0,E1 0.0,E2 0.0,E3 0.0,E4 0.0,E5 0.0,E6 0.0}
DECL FDAT Fswp_60_5474={TOOL_NO 2,BASE_NO 1,IPO_FRAME #BASE,POINT2[] " "}
DECL SPOT_TYPE SS_OLP32={GUN 2,PAIR #FIRST,RETR #CLO,CLO_TM 0,PGNO1 1,PRESS1 1.0,PGNO2 0,PRESS2 0.0}
DECL E6POS Xswp_60_5474={X 2110.28711,Y 855.671082,Z 456.949097,A 90.0540771,B 64.2556763,C -89.9835663,S 2,T 32,E1 0.0,E2 0.0,E3 0.0,E4 0.0,E5 0.0,E6 0.0}
DECL FDAT Fswp_60_5476={TOOL_NO 2,BASE_NO 1,IPO_FRAME #BASE,POINT2[] " "}
DECL SPOT_TYPE SS_OLP33={GUN 2,PAIR #FIRST,RETR #CLO,CLO_TM 0,PGNO1 1,PRESS1 1.0,PGNO2 0,PRESS2 0.0}
DECL E6POS Xswp_60_5476={X 2110.34009,Y 905.178589,Z 456.769592,A 90.0527725,B 64.2563324,C -89.9849319,S 2,T 32,E1 0.0,E2 0.0,E3 0.0,E4 0.0,E5 0.0,E6 0.0}
DECL FDAT Fp43={TOOL_NO 2,BASE_NO 1,IPO_FRAME #BASE,POINT2[] " "}
DECL PDAT PP_OLP51={VEL 100.0,ACC 100.0,APO_DIST 10.0,APO_MODE #CDIS}
DECL E6POS Xp43={X 2110.87891,Y 901.035706,Z 485.135986,A 90.0599365,B 64.2541199,C -89.9812317,S 2,T 32,E1 0.0,E2 0.0,E3 0.0,E4 0.0,E5 0.0,E6 0.0}
DECL FDAT Fp44={TOOL_NO 2,BASE_NO 1,IPO_FRAME #BASE,POINT2[] " "}
DECL PDAT PP_OLP52={VEL 100.0,ACC 100.0,APO_DIST 100.0,APO_MODE #CDIS}
DECL E6POS Xp44={X 2000.26196,Y 695.861572,Z 485.726196,A 89.9999924,B 70.0,C -90.0,S 2,T 32,E1 0.0,E2 0.0,E3 0.0,E4 0.0,E5 0.0,E6 0.0}
DECL FDAT Fp45={TOOL_NO 2,BASE_NO 1,IPO_FRAME #BASE,POINT2[] " "}
DECL E6POS Xp45={X 1640.98401,Y 593.222778,Z 2092.24194,A 121.9888,B 59.1547508,C -72.0102234,S 2,T 35,E1 0.0,E2 0.0,E3 0.0,E4 0.0,E5 0.0,E6 0.0}
DECL SPOT_SUGG_T LAST_SPOT={GUN[] "1                       ",RETR_CMD[] "#OPN                    ",CHOISE[] "#FIRST                  ",CLO_TM[] "1                       ",PGNO1[] "37                      ",PRESS1[] "0                       ",PGNO2[] "1                       ",PRESS2[] "0                       ",SPOT_PARAMS[] "NORMAL                  "}
DECL PDAT PPDAT1={VEL 100.0,ACC 100.0,APO_DIST 100.0}
DECL E6POS XSWP_60_5473={X 2137.86597,Y -862.153992,Z 452.227203,A -88.7343826,B 78.4225616,C 91.1146698,S 2,T 9,E1 0.0,E2 0.0,E3 0.0,E4 0.0,E5 0.0,E6 0.0}
DECL FDAT Fswp_60_5473={TOOL_NO 2,BASE_NO 1,IPO_FRAME #BASE,POINT2[] " ",TQ_STATE FALSE}
DECL PDAT PPDAT2={VEL 100.0,ACC 100.0,APO_DIST 100.0}
DECL PDAT PPDAT3={VEL 100.0,ACC 100.0,APO_DIST 100.0}
DECL PDAT PPDAT4={VEL 100.0,ACC 100.0,APO_DIST 100.0}
DECL PDAT PPDAT5={VEL 100.0,ACC 100.0,APO_DIST 100.0}
DECL PDAT PPDAT6={VEL 100.0,ACC 100.0,APO_DIST 100.0}
DECL PDAT PPDAT7={VEL 100.0,ACC 100.0,APO_DIST 100.0}
DECL PDAT PPDAT8={VEL 100.0,ACC 100.0,APO_DIST 100.0}
DECL PDAT PPDAT9={VEL 100.0,ACC 100.0,APO_DIST 100.0}
DECL PDAT PPDAT10={VEL 100.0,ACC 100.0,APO_DIST 100.0}
DECL PDAT PPDAT11={VEL 100.0,ACC 100.0,APO_DIST 100.0}
DECL PDAT PPDAT12={VEL 100.0,ACC 100.0,APO_DIST 100.0}
DECL PDAT PPDAT13={VEL 100.0,ACC 100.0,APO_DIST 100.0}
DECL PDAT PPDAT14={VEL 100.0,ACC 100.0,APO_DIST 100.0}
DECL PDAT PPDAT15={VEL 100.0,ACC 100.0,APO_DIST 100.0}
DECL PDAT PPDAT16={VEL 100.0,ACC 100.0,APO_DIST 100.0}
DECL PDAT PPDAT19={VEL 100.0,ACC 100.0,APO_DIST 100.0}
DECL PDAT PPDAT20={VEL 100.0,ACC 100.0,APO_DIST 100.0}
DECL PDAT PPDAT21={VEL 100.0,ACC 100.0,APO_DIST 100.0}
DECL PDAT PPDAT22={VEL 100.0,ACC 100.0,APO_DIST 100.0}
DECL PDAT PPDAT24={VEL 100.0,ACC 100.0,APO_DIST 100.0}
DECL PDAT PPDAT25={VEL 100.0,ACC 100.0,APO_DIST 100.0}
DECL PDAT PPDAT26={VEL 100.0,ACC 100.0,APO_DIST 100.0}
DECL PDAT PPDAT27={VEL 100.0,ACC 100.0,APO_DIST 100.0}
DECL PDAT PPDAT28={VEL 100.0,ACC 100.0,APO_DIST 100.0}
DECL PDAT PPDAT29={VEL 100.0,ACC 100.0,APO_DIST 100.0}
DECL PDAT PPDAT30={VEL 100.0,ACC 100.0,APO_DIST 100.0}
DECL PDAT PPDAT31={VEL 100.0,ACC 100.0,APO_DIST 100.0}
DECL PDAT PPDAT32={VEL 100.0,ACC 100.0,APO_DIST 100.0}
DECL PDAT PPDAT33={VEL 100.0,ACC 100.0,APO_DIST 100.0}
DECL PDAT PPDAT34={VEL 100.0,ACC 100.0,APO_DIST 100.0}
DECL PDAT PPDAT35={VEL 100.0,ACC 100.0,APO_DIST 100.0}
DECL LDAT LCPDAT1={VEL 2.0,ACC 100.0,APO_DIST 100.0,APO_FAC 50.0,AXIS_VEL 100.0,AXIS_ACC 100.0,ORI_TYP #VAR,CIRC_TYP #BASE,JERK_FAC 50.0,GEAR_JERK 50.0,EXAX_IGN 0}
DECL FDAT FHOME2={TOOL_NO 0,BASE_NO 0,IPO_FRAME #BASE,POINT2[] " ",TQ_STATE FALSE}
DECL E6POS XP1002={X 2124.38892,Y 154.860703,Z 481.495911,A -89.9889832,B 82.647049,C 90.0472488,S 2,T 0,E1 0.0,E2 0.0,E3 0.0,E4 0.0,E5 0.0,E6 0.0}
DECL FDAT Fp1002={TOOL_NO 2,BASE_NO 1,IPO_FRAME #BASE,POINT2[] " ",TQ_STATE FALSE}
DECL E6POS Xp1003={X 2133.75806,Y -97.5189972,Z 482.152191,A -90.0584869,B 82.6252213,C 89.9806213,S 2,T 9,E1 0.0,E2 0.0,E3 0.0,E4 0.0,E5 0.0,E6 0.0}
DECL FDAT Fp1003={TOOL_NO 2,BASE_NO 1,IPO_FRAME #BASE,POINT2[] " ",TQ_STATE FALSE}
DECL E6POS Xp1004={X 1992.92102,Y 52.5812416,Z 487.816101,A -90.0587463,B 82.6251678,C 89.9803238,S 2,T 8,E1 0.0,E2 0.0,E3 0.0,E4 0.0,E5 0.0,E6 0.0}
DECL FDAT Fp1004={TOOL_NO 2,BASE_NO 1,IPO_FRAME #BASE,POINT2[] " ",TQ_STATE FALSE}
DECL E6POS XP1005={X 2128.99097,Y -699.98407,Z 553.086487,A -89.4866867,B 67.1443481,C 90.4438095,S 2,T 9,E1 0.0,E2 0.0,E3 0.0,E4 0.0,E5 0.0,E6 0.0}
DECL FDAT Fp1005={TOOL_NO 2,BASE_NO 1,IPO_FRAME #BASE,POINT2[] " ",TQ_STATE FALSE}
DECL E6POS XP60_5441={X 2126.48706,Y -47.5520897,Z 457.337891,A 90.0909424,B 88.6400833,C -89.8710022,S 2,T 9,E1 0.0,E2 0.0,E3 0.0,E4 0.0,E5 0.0,E6 0.0}
DECL FDAT Fp60_5441={TOOL_NO 2,BASE_NO 1,IPO_FRAME #BASE,POINT2[] " ",TQ_STATE FALSE}
DECL E6POS XP6044={X 1992.97302,Y 101.959198,Z 481.442413,A -90.0514832,B 82.6261215,C 89.9883804,S 2,T 8,E1 0.0,E2 0.0,E3 0.0,E4 0.0,E5 0.0,E6 0.0}
DECL FDAT Fp6044={TOOL_NO 2,BASE_NO 1,IPO_FRAME #BASE,POINT2[] " ",TQ_STATE FALSE}
DECL PDAT PPDAT40={VEL 100.0,ACC 100.0,APO_DIST 100.0,APO_MODE #CDIS}
DECL E6POS XpFresa_05={X 1838.66003,Y 2546.56006,Z 4367.69092,A 105.045502,B -33.6448593,C -0.634051323,S 2,T 2,E1 0.0,E2 0.0,E3 0.0,E4 0.0,E5 0.0,E6 0.0}
DECL FDAT FpFresa_05={TOOL_NO 2,BASE_NO 1,IPO_FRAME #BASE,POINT2[] " ",TQ_STATE FALSE}
DECL PDAT PPDAT41={VEL 100.0,ACC 100.0,APO_DIST 100.0,APO_MODE #CDIS}
DECL E6POS XpFresa_06={X 4058.65503,Y 2091.6001,Z 4393.26904,A 52.5592613,B -34.2167282,C -0.74924773,S 2,T 2,E1 0.0,E2 0.0,E3 0.0,E4 0.0,E5 0.0,E6 0.0}
DECL FDAT FpFresa_06={TOOL_NO 2,BASE_NO 1,IPO_FRAME #BASE,POINT2[] " ",TQ_STATE FALSE}
DECL PDAT PPDAT42={VEL 100.0,ACC 100.0,APO_DIST 100.0,APO_MODE #CDIS}
DECL E6POS XpFresa_07={X 4058.65503,Y 2091.6001,Z 4393.26904,A 52.5592613,B -34.2167282,C -0.74924773,S 2,T 2,E1 0.0,E2 0.0,E3 0.0,E4 0.0,E5 0.0,E6 0.0}
DECL FDAT FpFresa_07={TOOL_NO 2,BASE_NO 1,IPO_FRAME #BASE,POINT2[] " ",TQ_STATE FALSE}
DECL PDAT PPDAT43={VEL 100.0,ACC 100.0,APO_DIST 100.0,APO_MODE #CDIS}
DECL E6POS XpFresa_08={X 1838.66003,Y 2546.56006,Z 4367.69092,A 105.045502,B -33.6448593,C -0.634051323,S 2,T 2,E1 0.0,E2 0.0,E3 0.0,E4 0.0,E5 0.0,E6 0.0}
DECL FDAT FpFresa_08={TOOL_NO 2,BASE_NO 1,IPO_FRAME #BASE,POINT2[] " ",TQ_STATE FALSE}
DECL PDAT PPDAT44={VEL 100.0,ACC 100.0,APO_DIST 100.0,APO_MODE #CDIS}
DECL E6POS XpFresa_01={X 1838.66003,Y 2546.56006,Z 4367.69092,A 105.045502,B -33.6448593,C -0.634051323,S 2,T 2,E1 0.0,E2 0.0,E3 0.0,E4 0.0,E5 0.0,E6 0.0}
DECL FDAT FpFresa_01={TOOL_NO 2,BASE_NO 1,IPO_FRAME #BASE,POINT2[] " ",TQ_STATE FALSE}
DECL PDAT PPDAT45={VEL 100.0,ACC 100.0,APO_DIST 100.0,APO_MODE #CDIS}
DECL E6POS XpFresa_02={X 4058.65503,Y 2091.6001,Z 4393.26904,A 52.5592613,B -34.2167282,C -0.74924773,S 2,T 2,E1 0.0,E2 0.0,E3 0.0,E4 0.0,E5 0.0,E6 0.0}
DECL FDAT FpFresa_02={TOOL_NO 2,BASE_NO 1,IPO_FRAME #BASE,POINT2[] " ",TQ_STATE FALSE}
DECL PDAT PPDAT46={VEL 100.0,ACC 100.0,APO_DIST 100.0,APO_MODE #CDIS}
DECL E6POS XpFresa_03={X 4058.65503,Y 2091.6001,Z 4393.26904,A 52.5592613,B -34.2167282,C -0.74924773,S 2,T 2,E1 0.0,E2 0.0,E3 0.0,E4 0.0,E5 0.0,E6 0.0}
DECL FDAT FpFresa_03={TOOL_NO 2,BASE_NO 1,IPO_FRAME #BASE,POINT2[] " ",TQ_STATE FALSE}
DECL PDAT PPDAT47={VEL 100.0,ACC 100.0,APO_DIST 100.0,APO_MODE #CDIS}
DECL E6POS XpFresa_04={X 1838.66003,Y 2546.56006,Z 4367.69092,A 105.045502,B -33.6448593,C -0.634051323,S 2,T 2,E1 0.0,E2 0.0,E3 0.0,E4 0.0,E5 0.0,E6 0.0}
DECL FDAT FpFresa_04={TOOL_NO 2,BASE_NO 1,IPO_FRAME #BASE,POINT2[] " ",TQ_STATE FALSE}
DECL E6POS XP6045={X 2137.41992,Y -896.906128,Z 484.981689,A -90.0024567,B 55.4039993,C 89.9980087,S 2,T 9,E1 0.0,E2 0.0,E3 0.0,E4 0.0,E5 0.0,E6 0.0}
DECL FDAT Fp6045={TOOL_NO 2,BASE_NO 1,IPO_FRAME #BASE,POINT2[] " ",TQ_STATE FALSE}
DECL PDAT PPDAT48={VEL 100.0,ACC 100.0,APO_DIST 100.0,APO_MODE #CDIS}
DECL E6POS XP6046={X 2125.552,Y 250.760696,Z 488.898499,A -89.462883,B 88.9658203,C 90.4861526,S 2,T 0,E1 0.0,E2 0.0,E3 0.0,E4 0.0,E5 0.0,E6 0.0}
DECL FDAT Fp6046={TOOL_NO 2,BASE_NO 1,IPO_FRAME #BASE,POINT2[] " ",TQ_STATE FALSE}
DECL PDAT PPDAT49={VEL 100.0,ACC 100.0,APO_DIST 10.0,APO_MODE #CDIS}
DECL PDAT PPDAT51={VEL 100.0,ACC 100.0,APO_DIST 100.0,APO_MODE #CDIS}
DECL E6POS XP6049={X 2068.2439,Y 260.153015,Z 493.036407,A -88.7928772,B 89.0078278,C 91.1528473,S 2,T 0,E1 0.0,E2 0.0,E3 0.0,E4 0.0,E5 0.0,E6 0.0}
DECL FDAT Fp6049={TOOL_NO 2,BASE_NO 1,IPO_FRAME #BASE,POINT2[] " ",TQ_STATE FALSE}
DECL PDAT PPDAT52={VEL 100.0,ACC 100.0,APO_DIST 100.0,APO_MODE #CDIS}
DECL E6POS XP6050={X 2066.41211,Y 467.441589,Z 488.970886,A -91.4706802,B 89.0215607,C 88.4768829,S 2,T 0,E1 0.0,E2 0.0,E3 0.0,E4 0.0,E5 0.0,E6 0.0}
DECL FDAT Fp6050={TOOL_NO 2,BASE_NO 1,IPO_FRAME #BASE,POINT2[] " ",TQ_STATE FALSE}
DECL PDAT PPDAT53={VEL 100.0,ACC 100.0,APO_DIST 100.0,APO_MODE #CDIS}
DECL E6POS XP6051={X 2124.6189,Y 469.901886,Z 484.399597,A -91.5506821,B 89.0213776,C 88.396843,S 2,T 0,E1 0.0,E2 0.0,E3 0.0,E4 0.0,E5 0.0,E6 0.0}
DECL FDAT Fp6051={TOOL_NO 2,BASE_NO 1,IPO_FRAME #BASE,POINT2[] " ",TQ_STATE FALSE}
DECL PDAT PPDAT54={VEL 100.0,ACC 100.0,APO_DIST 100.0,APO_MODE #CDIS}
DECL E6POS XSWP_60_5497={X 2126.5459,Y 8.33220863,Z 456.357788,A 90.0595322,B 88.6408386,C -89.9031372,S 2,T 9,E1 0.0,E2 0.0,E3 0.0,E4 0.0,E5 0.0,E6 0.0}
DECL FDAT Fswp_60_5497={TOOL_NO 2,BASE_NO 1,IPO_FRAME #BASE,POINT2[] " ",TQ_STATE FALSE}
DECL PDAT PPDAT55={VEL 100.0,ACC 100.0,APO_DIST 100.0,APO_MODE #CDIS}
DECL PDAT PP_OLP55={VEL 100.0,ACC 100.0,APO_DIST 0.0}
DECL E6POS Xswp_60_5477={X 2137.69897,Y -795.659485,Z 457.93811,A -90.1632385,B 69.9812317,C 89.8293381,S 2,T 9,E1 0.0,E2 0.0,E3 0.0,E4 0.0,E5 0.0,E6 0.0}
DECL FDAT Fswp_60_5477={TOOL_NO 2,BASE_NO 1,IPO_FRAME #BASE,POINT2[] " "}
DECL PDAT PP_OLP56={VEL 100.0,ACC 100.0,APO_DIST 0.0}
DECL E6POS Xswp_60_5478={X 2122.81396,Y 313.206909,Z 456.674713,A 89.9989166,B 64.9993362,C -90.000679,S 2,T 33,E1 0.0,E2 0.0,E3 0.0,E4 0.0,E5 0.0,E6 0.0}
DECL FDAT Fswp_60_5478={TOOL_NO 2,BASE_NO 1,IPO_FRAME #BASE,POINT2[] " ",TQ_STATE FALSE}
DECL E6POS XP5={X 814.125122,Y 41.8001404,Z 3106.80591,A -178.988495,B 40.6093903,C 0.315513402,S 2,T 2,E1 0.0,E2 0.0,E3 0.0,E4 0.0,E5 0.0,E6 0.0}
DECL FDAT FP5={TOOL_NO 2,BASE_NO 1,IPO_FRAME #BASE,POINT2[] " ",TQ_STATE FALSE}
DECL PDAT PPDAT56={VEL 100.0,ACC 100.0,APO_DIST 5.0,APO_MODE #CDIS}
DECL E6POS XP6={X 814.12439,Y 41.8147888,Z 3106.82007,A -178.988297,B 40.608551,C 0.315220714,S 2,T 2,E1 0.0,E2 0.0,E3 0.0,E4 0.0,E5 0.0,E6 0.0}
DECL FDAT FP6={TOOL_NO 2,BASE_NO 1,IPO_FRAME #BASE,POINT2[] " ",TQ_STATE FALSE}
DECL PDAT PPDAT57={VEL 100.0,ACC 100.0,APO_DIST 5.0,APO_MODE #CDIS}
DECL E6POS XP7={X 2309.73291,Y 2488.5769,Z 4622.88818,A 56.7310791,B -23.3806591,C 61.3704605,S 2,T 42,E1 0.0,E2 0.0,E3 0.0,E4 0.0,E5 0.0,E6 0.0}
DECL FDAT FP7={TOOL_NO 2,BASE_NO 1,IPO_FRAME #BASE,POINT2[] " ",TQ_STATE FALSE}
DECL PDAT PPDAT58={VEL 100.0,ACC 100.0,APO_DIST 5.0,APO_MODE #CDIS}
DECL E6POS XP8={X 2114.68311,Y 828.082092,Z 456.497803,A 90.042717,B 73.3173523,C -89.9860916,S 2,T 32,E1 0.0,E2 0.0,E3 0.0,E4 0.0,E5 0.0,E6 0.0}
DECL FDAT FP8={TOOL_NO 2,BASE_NO 1,IPO_FRAME #BASE,POINT2[] " ",TQ_STATE FALSE}
DECL PDAT PPDAT59={VEL 100.0,ACC 100.0,APO_DIST 5.0,APO_MODE #CDIS}
ENDDAT
